KUKA KRL program: MyProgram_322().src

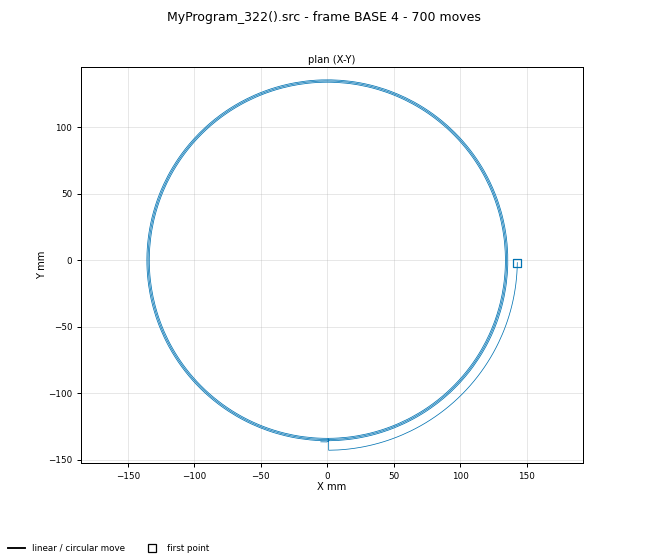
[picture p0: tool path of MyProgram_322().src in frame BASE 4, 700 of 700 moves have a stored position in this frame; points joined in program order, loops and branches not executed]
&ACCESS RVP
&REL 1
&PARAM TEMPLATE = C:\KRC\Roboter\Template\vorgabe
&PARAM EDITMASK = *
DEF MyProgram_322()
; ---- Setting reference (Base) ----
$BASE = BASE_DATA[4]

; --------------------------
; ---- Setting tool (TCP) ----
$TOOL = TOOL_DATA[3]
; --------------------------

$VEL.CP = VEL_APROX_PRINT
Startdeposition()
$VEL.CP = VEL_PRINT
LIN {X 142.7599,Y -1.7436,Z 185,A 2.3908,B 3.1922,C 0.193,E1 3.3578,E2 451.0051} C_DIS
LIN {X 142.6356,Y -6.2063,Z 185,A 0.7116,B 3.1919,C 0.1969,E1 3.3576,E2 452.6705} C_DIS
LIN {X 142.4407,Y -9.7017,Z 185,A -0.6684,B 3.1917,C 0.2006,E1 3.3574,E2 454.0481} C_DIS
LIN {X 142.1591,Y -13.1909,Z 185,A -2.1332,B 3.1914,C 0.2052,E1 3.357,E2 455.5219} C_DIS
LIN {X 141.6977,Y -17.466,Z 185,A -3.6398,B 3.1913,C 0.2077,E1 3.3566,E2 457.0004} C_DIS
LIN {X 141.2248,Y -20.9551,Z 185,A -4.9961,B 3.191,C 0.211,E1 3.356,E2 458.3501} C_DIS
LIN {X 140.669,Y -24.408,Z 185,A -6.3574,B 3.1908,C 0.2145,E1 3.3554,E2 459.7068} C_DIS
LIN {X 140.0285,Y -27.8456,Z 185,A -7.6988,B 3.1906,C 0.2178,E1 3.3547,E2 461.0409} C_DIS
LIN {X 139.3005,Y -31.2823,Z 185,A -9.0472,B 3.1904,C 0.221,E1 3.3539,E2 462.382} C_DIS
LIN {X 138.4934,Y -34.68,Z 185,A -10.3892,B 3.1901,C 0.2242,E1 3.353,E2 463.717} C_DIS
LIN {X 137.5957,Y -38.0853,Z 185,A -11.7403,B 3.1899,C 0.2274,E1 3.3521,E2 465.0608} C_DIS
LIN {X 136.4692,Y -41.9415,Z 185,A -13.3324,B 3.1896,C 0.2316,E1 3.3508,E2 466.6513} C_DIS
LIN {X 135.3217,Y -45.5096,Z 185,A -14.7313,B 3.1894,C 0.2346,E1 3.3496,E2 468.0371} C_DIS
LIN {X 134.1171,Y -48.9469,Z 185,A -16.135,B 3.1892,C 0.2379,E1 3.3483,E2 469.4342} C_DIS
LIN {X 132.912,Y -52.1294,Z 185,A -17.4464,B 3.1889,C 0.2409,E1 3.3469,E2 470.7393} C_DIS
LIN {X 131.5372,Y -55.5078,Z 185,A -18.8532,B 3.1887,C 0.2442,E1 3.3455,E2 472.1395} C_DIS
LIN {X 130.1671,Y -58.6477,Z 185,A -20.1759,B 3.1884,C 0.2472,E1 3.344,E2 473.4562} C_DIS
LIN {X 128.7579,Y -61.6788,Z 185,A -21.4838,B 3.1882,C 0.2503,E1 3.3424,E2 474.7605} C_DIS
LIN {X 126.9178,Y -65.3849,Z 185,A -23.0872,B 3.1879,C 0.254,E1 3.3404,E2 476.3576} C_DIS
LIN {X 124.8595,Y -69.2355,Z 185,A -24.7994,B 3.1876,C 0.258,E1 3.3381,E2 478.0657} C_DIS
LIN {X 122.6632,Y -73.0559,Z 185,A -26.5049,B 3.1873,C 0.2617,E1 3.3357,E2 479.7641} C_DIS
LIN {X 120.4066,Y -76.7189,Z 185,A -28.1924,B 3.187,C 0.2655,E1 3.3332,E2 481.4476} C_DIS
LIN {X 117.9943,Y -80.3801,Z 185,A -29.8939,B 3.1867,C 0.2692,E1 3.3306,E2 483.1427} C_DIS
LIN {X 115.4359,Y -84.0122,Z 185,A -31.5557,B 3.1864,C 0.2721,E1 3.3279,E2 484.7893} C_DIS
LIN {X 112.8442,Y -87.4622,Z 185,A -33.2618,B 3.1861,C 0.2758,E1 3.325,E2 486.4933} C_DIS
LIN {X 110.1935,Y -90.7797,Z 185,A -34.9543,B 3.1858,C 0.2796,E1 3.3221,E2 488.1855} C_DIS
LIN {X 107.2025,Y -94.293,Z 185,A -36.7037,B 3.1855,C 0.2826,E1 3.3189,E2 489.9224} C_DIS
LIN {X 104.325,Y -97.4668,Z 185,A -38.3639,B 3.1852,C 0.2857,E1 3.3158,E2 491.5759} C_DIS
LIN {X 101.2534,Y -100.6538,Z 185,A -40.0668,B 3.185,C 0.2887,E1 3.3124,E2 493.2702} C_DIS
LIN {X 98.1844,Y -103.65,Z 185,A -41.7616,B 3.1847,C 0.292,E1 3.309,E2 494.9627} C_DIS
LIN {X 94.9103,Y -106.6568,Z 185,A -43.4985,B 3.1844,C 0.295,E1 3.3054,E2 496.6945} C_DIS
LIN {X 91.5632,Y -109.5431,Z 185,A -45.1906,B 3.1841,C 0.2977,E1 3.3019,E2 498.3768} C_DIS
LIN {X 88.2302,Y -112.2447,Z 185,A -46.8727,B 3.1839,C 0.3005,E1 3.2982,E2 500.0548} C_DIS
LIN {X 84.7543,Y -114.8922,Z 185,A -48.591,B 3.1836,C 0.3033,E1 3.2944,E2 501.7696} C_DIS
LIN {X 81.1633,Y -117.457,Z 185,A -50.3222,B 3.1833,C 0.306,E1 3.2904,E2 503.4967} C_DIS
LIN {X 77.4935,Y -119.9095,Z 185,A -52.0213,B 3.1831,C 0.3082,E1 3.2865,E2 505.1871} C_DIS
LIN {X 73.8618,Y -122.1797,Z 185,A -53.6994,B 3.1829,C 0.3106,E1 3.2825,E2 506.8609} C_DIS
LIN {X 70.0297,Y -124.4158,Z 185,A -55.4462,B 3.1827,C 0.313,E1 3.2783,E2 508.6043} C_DIS
LIN {X 66.174,Y -126.5065,Z 185,A -57.1052,B 3.1825,C 0.3146,E1 3.2742,E2 510.2505} C_DIS
LIN {X 62.6225,Y -128.3029,Z 185,A -58.6591,B 3.1823,C 0.3164,E1 3.2703,E2 511.7996} C_DIS
LIN {X 59.4743,Y -129.7918,Z 185,A -59.9839,B 3.1823,C 0.3176,E1 3.267,E2 513.1153} C_DIS
LIN {X 56.3886,Y -131.1613,Z 185,A -61.3699,B 3.182,C 0.3196,E1 3.2634,E2 514.5065} C_DIS
LIN {X 52.762,Y -132.6631,Z 185,A -62.9943,B 3.1818,C 0.3219,E1 3.2592,E2 516.1389} C_DIS
LIN {X 48.9995,Y -134.0981,Z 185,A -64.5241,B 3.1817,C 0.323,E1 3.2552,E2 517.6578} C_DIS
LIN {X 45.7133,Y -135.2538,Z 185,A -65.8658,B 3.1816,C 0.324,E1 3.2517,E2 518.9926} C_DIS
LIN {X 42.3516,Y -136.3437,Z 185,A -67.3012,B 3.1814,C 0.3255,E1 3.2479,E2 520.4313} C_DIS
LIN {X 38.837,Y -137.3854,Z 185,A -68.8442,B 3.1812,C 0.3275,E1 3.2437,E2 521.9853} C_DIS
LIN {X 34.6802,Y -138.4934,Z 185,A -70.406,B 3.1812,C 0.3275,E1 3.2395,E2 523.5252} C_DIS
LIN {X 31.4204,Y -139.2689,Z 185,A -71.7456,B 3.1811,C 0.3286,E1 3.2359,E2 524.865} C_DIS
LIN {X 27.8611,Y -140.0253,Z 185,A -73.1737,B 3.1811,C 0.3294,E1 3.232,E2 526.2895} C_DIS
LIN {X 24.4235,Y -140.6662,Z 185,A -74.5592,B 3.1809,C 0.3302,E1 3.2282,E2 527.6734} C_DIS
LIN {X 20.03,Y -141.357,Z 185,A -76.38,B 3.1808,C 0.3315,E1 3.2231,E2 529.5001} C_DIS
LIN {X 15.7373,Y -141.8997,Z 185,A -78.0703,B 3.1808,C 0.332,E1 3.2184,E2 531.185} C_DIS
LIN {X 11.4541,Y -142.3099,Z 185,A -79.7619,B 3.1807,C 0.3324,E1 3.2137,E2 532.8726} C_DIS
LIN {X 7.9599,Y -142.5492,Z 185,A -81.1954,B 3.1807,C 0.3331,E1 3.2097,E2 534.3107} C_DIS
LIN {X 4.3071,Y -142.7045,Z 185,A -82.7592,B 3.1805,C 0.3343,E1 3.2053,E2 535.8887} C_DIS
LIN {X 1.005,Y -142.7647,Z 185,A -83.6736,B 3.1808,C 0.3313,E1 3.2029,E2 536.7463} C_DIS
Enddeposition()
LIN {X 0.9687,Y -133.816,Z 186,A -83.71,B 3.076,C 0.3108,E1 3.0971,E2 536.5076} C_DIS
Startdeposition()
$VEL.CP = VEL_PRINT
LIN {X 4.436,Y -133.7511,Z 186,A -81.8774,B 3.0763,C 0.3079,E1 3.1024,E2 534.6292} C_DIS
LIN {X 8.1929,Y -133.5716,Z 186,A -80.4113,B 3.0763,C 0.3084,E1 3.1064,E2 533.1809} C_DIS
LIN {X 11.4617,Y -133.331,Z 186,A -79.0228,B 3.0763,C 0.308,E1 3.1103,E2 531.7937} C_DIS
LIN {X 14.751,Y -133.0078,Z 186,A -77.6221,B 3.0763,C 0.3074,E1 3.1142,E2 530.394} C_DIS
LIN {X 18.5236,Y -132.5349,Z 186,A -75.9557,B 3.0765,C 0.3063,E1 3.1188,E2 528.7217} C_DIS
LIN {X 22.8645,Y -131.8567,Z 186,A -74.1261,B 3.0765,C 0.3055,E1 3.1238,E2 526.8978} C_DIS
LIN {X 26.0898,Y -131.2559,Z 186,A -72.7336,B 3.0766,C 0.3046,E1 3.1277,E2 525.506} C_DIS
LIN {X 29.3206,Y -130.5717,Z 186,A -71.3456,B 3.0767,C 0.3038,E1 3.1314,E2 524.1205} C_DIS
LIN {X 32.5132,Y -129.8133,Z 186,A -69.9613,B 3.0768,C 0.3028,E1 3.1352,E2 522.738} C_DIS
LIN {X 36.191,Y -128.8357,Z 186,A -68.2956,B 3.077,C 0.301,E1 3.1397,E2 521.0665} C_DIS
LIN {X 40.4049,Y -127.5772,Z 186,A -66.502,B 3.0771,C 0.2999,E1 3.1445,E2 519.2834} C_DIS
LIN {X 43.5438,Y -126.5402,Z 186,A -65.1143,B 3.0772,C 0.2986,E1 3.1481,E2 517.8983} C_DIS
LIN {X 47.1263,Y -125.2499,Z 186,A -63.5124,B 3.0774,C 0.297,E1 3.1523,E2 516.299} C_DIS
LIN {X 50.1812,Y -124.0574,Z 186,A -62.1351,B 3.0775,C 0.2956,E1 3.1559,E2 514.9243} C_DIS
LIN {X 53.7484,Y -122.556,Z 186,A -60.3934,B 3.0778,C 0.2928,E1 3.1604,E2 513.1704} C_DIS
LIN {X 57.6835,Y -120.7517,Z 186,A -58.6987,B 3.0778,C 0.2917,E1 3.1646,E2 511.495} C_DIS
LIN {X 60.1603,Y -119.5386,Z 186,A -57.5521,B 3.078,C 0.2903,E1 3.1675,E2 510.3521} C_DIS
LIN {X 63.3281,Y -117.8917,Z 186,A -56.1166,B 3.0781,C 0.2889,E1 3.171,E2 508.9276} C_DIS
LIN {X 66.3957,Y -116.1917,Z 186,A -54.5879,B 3.0784,C 0.2864,E1 3.1748,E2 507.3942} C_DIS
LIN {X 69.1892,Y -114.5502,Z 186,A -53.1474,B 3.0786,C 0.2838,E1 3.1782,E2 505.9457} C_DIS
LIN {X 72.8586,Y -112.252,Z 186,A -51.3975,B 3.0788,C 0.2817,E1 3.1823,E2 504.2079} C_DIS
LIN {X 76.0934,Y -110.0857,Z 186,A -49.6753,B 3.0791,C 0.2783,E1 3.1863,E2 502.4773} C_DIS
LIN {X 79.7248,Y -107.4845,Z 186,A -47.845,B 3.0794,C 0.2757,E1 3.1904,E2 500.6562} C_DIS
LIN {X 83.1812,Y -104.8324,Z 186,A -46.0377,B 3.0796,C 0.2728,E1 3.1944,E2 498.8549} C_DIS
LIN {X 86.574,Y -102.0483,Z 186,A -44.2223,B 3.0799,C 0.2698,E1 3.1983,E2 497.0463} C_DIS
LIN {X 89.8778,Y -99.1508,Z 186,A -42.4453,B 3.0801,C 0.267,E1 3.202,E2 495.2813} C_DIS
LIN {X 92.8686,Y -96.3556,Z 186,A -40.7416,B 3.0804,C 0.2639,E1 3.2054,E2 493.5826} C_DIS
LIN {X 95.7716,Y -93.4709,Z 186,A -38.9685,B 3.0807,C 0.2601,E1 3.2089,E2 491.8054} C_DIS
LIN {X 98.7809,Y -90.2849,Z 186,A -37.1738,B 3.081,C 0.2568,E1 3.2123,E2 490.0196} C_DIS
LIN {X 101.6976,Y -86.9865,Z 186,A -35.4113,B 3.0812,C 0.2538,E1 3.2155,E2 488.2715} C_DIS
LIN {X 104.127,Y -84.0623,Z 186,A -33.8119,B 3.0815,C 0.2504,E1 3.2183,E2 486.6744} C_DIS
LIN {X 106.8292,Y -80.6004,Z 186,A -31.9916,B 3.0818,C 0.2466,E1 3.2214,E2 484.8602} C_DIS
LIN {X 109.4259,Y -77.0383,Z 186,A -30.1807,B 3.0821,C 0.2429,E1 3.2243,E2 483.0577} C_DIS
LIN {X 111.8951,Y -73.406,Z 186,A -28.3662,B 3.0824,C 0.239,E1 3.2272,E2 481.2502} C_DIS
LIN {X 113.9323,Y -70.2026,Z 186,A -26.9035,B 3.0826,C 0.2366,E1 3.2293,E2 479.8069} C_DIS
LIN {X 115.8253,Y -67.0328,Z 186,A -25.3615,B 3.0829,C 0.2331,E1 3.2315,E2 478.2686} C_DIS
LIN {X 117.4797,Y -64.0892,Z 186,A -23.9557,B 3.0831,C 0.2299,E1 3.2334,E2 476.8668} C_DIS
LIN {X 119.0131,Y -61.1926,Z 186,A -22.6488,B 3.0833,C 0.2272,E1 3.235,E2 475.571} C_DIS
LIN {X 120.2635,Y -58.6973,Z 186,A -21.492,B 3.0835,C 0.2245,E1 3.2365,E2 474.4182} C_DIS
LIN {X 121.6664,Y -55.7303,Z 186,A -20.0767,B 3.0838,C 0.2208,E1 3.2381,E2 473.0004} C_DIS
LIN {X 123.431,Y -51.7028,Z 186,A -18.256,B 3.0841,C 0.2165,E1 3.2401,E2 471.1861} C_DIS
LIN {X 124.9906,Y -47.8147,Z 186,A -16.4578,B 3.0844,C 0.2117,E1 3.242,E2 469.386} C_DIS
LIN {X 126.1657,Y -44.6236,Z 186,A -15.0773,B 3.0846,C 0.2085,E1 3.2432,E2 468.014} C_DIS
LIN {X 127.5813,Y -40.3922,Z 186,A -13.3493,B 3.0849,C 0.2051,E1 3.2447,E2 466.3077} C_DIS
LIN {X 128.8337,Y -36.1982,Z 186,A -11.5227,B 3.0852,C 0.2005,E1 3.2461,E2 464.4856} C_DIS
LIN {X 129.9409,Y -32.0037,Z 186,A -9.8212,B 3.0854,C 0.1969,E1 3.2473,E2 462.8025} C_DIS
LIN {X 130.6882,Y -28.7984,Z 186,A -8.4768,B 3.0856,C 0.1937,E1 3.2481,E2 461.4653} C_DIS
LIN {X 131.3542,Y -25.5879,Z 186,A -7.1334,B 3.0858,C 0.1904,E1 3.2489,E2 460.1284} C_DIS
LIN {X 131.9414,Y -22.3615,Z 186,A -5.9696,B 3.0859,C 0.1888,E1 3.2494,E2 458.9938} C_DIS
LIN {X 132.3756,Y -19.6384,Z 186,A -4.5318,B 3.0863,C 0.183,E1 3.25,E2 457.5229} C_DIS
LIN {X 132.8782,Y -15.8696,Z 186,A -3.1128,B 3.0863,C 0.1805,E1 3.2505,E2 456.1289} C_DIS
LIN {X 133.2421,Y -12.4557,Z 186,A -1.7289,B 3.0866,C 0.1772,E1 3.2509,E2 454.7548} C_DIS
LIN {X 133.4983,Y -9.3201,Z 186,A -0.4325,B 3.0868,C 0.1739,E1 3.2512,E2 453.4639} C_DIS
LIN {X 133.7115,Y -5.4589,Z 186,A 1.2482,B 3.087,C 0.169,E1 3.2514,E2 451.7789} C_DIS
LIN {X 133.8137,Y -1.6575,Z 186,A 2.6544,B 3.0872,C 0.1666,E1 3.2514,E2 450.3995} C_DIS
LIN {X 133.805,Y 2.1748,Z 186,A 4.3608,B 3.0875,C 0.1613,E1 3.2514,E2 448.6837} C_DIS
LIN {X 133.6617,Y 6.5635,Z 186,A 6.0882,B 3.0877,C 0.1575,E1 3.2512,E2 446.9743} C_DIS
LIN {X 133.4607,Y 9.8358,Z 186,A 7.4615,B 3.0878,C 0.1539,E1 3.251,E2 445.6039} C_DIS
LIN {X 133.1787,Y 13.1156,Z 186,A 8.766,B 3.088,C 0.1509,E1 3.2506,E2 444.3115} C_DIS
LIN {X 132.8167,Y 16.3854,Z 186,A 10.2269,B 3.0882,C 0.1465,E1 3.2502,E2 442.8433} C_DIS
LIN {X 132.2965,Y 20.154,Z 186,A 11.5023,B 3.0882,C 0.1454,E1 3.2497,E2 441.6108} C_DIS
LIN {X 131.855,Y 22.8737,Z 186,A 12.8158,B 3.0885,C 0.1408,E1 3.2491,E2 440.2802} C_DIS
LIN {X 131.2542,Y 26.0985,Z 186,A 14.1611,B 3.0886,C 0.1375,E1 3.2484,E2 438.9414} C_DIS
LIN {X 130.571,Y 29.3235,Z 186,A 15.5046,B 3.0888,C 0.1343,E1 3.2476,E2 437.6055} C_DIS
LIN {X 129.8121,Y 32.5177,Z 186,A 16.8476,B 3.0888,C 0.131,E1 3.2467,E2 436.2695} C_DIS
LIN {X 128.8341,Y 36.1967,Z 186,A 18.466,B 3.0891,C 0.1267,E1 3.2455,E2 434.6516} C_DIS
LIN {X 127.5731,Y 40.418,Z 186,A 20.3118,B 3.0893,C 0.122,E1 3.244,E2 432.81} C_DIS
LIN {X 126.1683,Y 44.6162,Z 186,A 22.1632,B 3.0894,C 0.1173,E1 3.2423,E2 430.9631} C_DIS
LIN {X 124.6797,Y 48.6144,Z 186,A 23.7847,B 3.0895,C 0.1145,E1 3.2407,E2 429.366} C_DIS
LIN {X 123.4332,Y 51.6976,Z 186,A 25.2113,B 3.0897,C 0.1107,E1 3.2392,E2 427.9385} C_DIS
LIN {X 121.6698,Y 55.723,Z 186,A 27.062,B 3.0898,C 0.1061,E1 3.2371,E2 426.0909} C_DIS
LIN {X 120.0375,Y 59.1553,Z 186,A 28.3574,B 3.0898,C 0.1051,E1 3.2355,E2 424.8353} C_DIS
LIN {X 118.7857,Y 61.634,Z 186,A 29.6269,B 3.09,C 0.1013,E1 3.2339,E2 423.5556} C_DIS
LIN {X 117.2392,Y 64.529,Z 186,A 31.1268,B 3.0901,C 0.0969,E1 3.2319,E2 422.0437} C_DIS
LIN {X 115.3504,Y 67.8467,Z 186,A 32.5705,B 3.0902,C 0.0947,E1 3.2299,E2 420.6227} C_DIS
LIN {X 113.3422,Y 71.1516,Z 186,A 34.2658,B 3.0903,C 0.0903,E1 3.2274,E2 418.922} C_DIS
LIN {X 111.2743,Y 74.3434,Z 186,A 35.729,B 3.0904,C 0.0879,E1 3.2252,E2 417.4784} C_DIS
LIN {X 109.4199,Y 77.0468,Z 186,A 37.1703,B 3.0905,C 0.0843,E1 3.2229,E2 416.0322} C_DIS
LIN {X 106.8195,Y 80.6133,Z 186,A 39.0047,B 3.0906,C 0.0805,E1 3.2198,E2 414.2041} C_DIS
LIN {X 103.9631,Y 84.2655,Z 186,A 40.926,B 3.0907,C 0.0766,E1 3.2165,E2 412.29} C_DIS
LIN {X 101.1608,Y 87.61,Z 186,A 42.7319,B 3.0908,C 0.073,E1 3.2132,E2 410.4913} C_DIS
LIN {X 98.4298,Y 90.6669,Z 186,A 44.4122,B 3.0908,C 0.07,E1 3.2101,E2 408.8197} C_DIS
LIN {X 95.582,Y 93.6641,Z 186,A 46.1113,B 3.0909,C 0.0669,E1 3.2068,E2 407.1289} C_DIS
LIN {X 92.473,Y 96.7349,Z 186,A 47.8811,B 3.091,C 0.064,E1 3.2033,E2 405.371} C_DIS
LIN {X 89.6931,Y 99.3184,Z 186,A 49.5251,B 3.091,C 0.0606,E1 3.1999,E2 403.7246} C_DIS
LIN {X 86.5877,Y 102.0367,Z 186,A 51.2202,B 3.0911,C 0.0579,E1 3.1963,E2 402.0379} C_DIS
LIN {X 83.1898,Y 104.8255,Z 186,A 53.0445,B 3.0911,C 0.0549,E1 3.1924,E2 400.2205} C_DIS
LIN {X 79.7194,Y 107.4885,Z 186,A 54.8692,B 3.0912,C 0.052,E1 3.1883,E2 398.4015} C_DIS
LIN {X 76.2646,Y 109.9666,Z 186,A 56.4511,B 3.0912,C 0.0509,E1 3.1848,E2 396.8481} C_DIS
LIN {X 73.4139,Y 111.8899,Z 186,A 58.0702,B 3.0913,C 0.0473,E1 3.181,E2 395.2115} C_DIS
LIN {X 70.2047,Y 113.931,Z 186,A 59.555,B 3.0913,C 0.0459,E1 3.1775,E2 393.7439} C_DIS
LIN {X 67.3921,Y 115.6173,Z 186,A 61.0498,B 3.0913,C 0.043,E1 3.1739,E2 392.2383} C_DIS
LIN {X 64.0999,Y 117.4739,Z 186,A 62.5393,B 3.0913,C 0.0417,E1 3.1703,E2 390.7642} C_DIS
LIN {X 61.1645,Y 119.0273,Z 186,A 63.7829,B 3.0913,C 0.0411,E1 3.1672,E2 389.542} C_DIS
LIN {X 58.6915,Y 120.2663,Z 186,A 65.0633,B 3.0914,C 0.0388,E1 3.164,E2 388.2503} C_DIS
LIN {X 55.7246,Y 121.6691,Z 186,A 66.5094,B 3.0914,C 0.0367,E1 3.1603,E2 386.7994} C_DIS
LIN {X 51.6992,Y 123.4325,Z 186,A 68.3671,B 3.0914,C 0.0346,E1 3.1555,E2 384.9448} C_DIS
LIN {X 48.1677,Y 124.8534,Z 186,A 69.8792,B 3.0914,C 0.0336,E1 3.1516,E2 383.447} C_DIS
LIN {X 44.6082,Y 126.1712,Z 186,A 71.6386,B 3.0915,C 0.0309,E1 3.147,E2 381.6721} C_DIS
LIN {X 40.9108,Y 127.4156,Z 186,A 72.9052,B 3.0915,C 0.0323,E1 3.1437,E2 380.4535} C_DIS
LIN {X 38.341,Y 128.2145,Z 186,A 74.4123,B 3.0915,C 0.0286,E1 3.1396,E2 378.9047} C_DIS
LIN {X 34.1077,Y 129.4034,Z 186,A 76.1827,B 3.0915,C 0.0278,E1 3.1349,E2 377.1481} C_DIS
LIN {X 30.4151,Y 130.3217,Z 186,A 77.7251,B 3.0915,C 0.0271,E1 3.1307,E2 375.6164} C_DIS
LIN {X 27.2108,Y 131.0279,Z 186,A 79.1175,B 3.0915,C 0.0262,E1 3.1269,E2 374.2259} C_DIS
LIN {X 23.9747,Y 131.658,Z 186,A 80.5085,B 3.0915,C 0.0255,E1 3.1231,E2 372.8377} C_DIS
LIN {X 21.261,Y 132.125,Z 186,A 81.6808,B 3.0915,C 0.0249,E1 3.1199,E2 371.6666} C_DIS
LIN {X 17.4962,Y 132.6739,Z 186,A 83.2879,B 3.0915,C 0.0242,E1 3.1154,E2 370.0626} C_DIS
LIN {X 14.2377,Y 133.063,Z 186,A 84.6779,B 3.0915,C 0.0237,E1 3.1116,E2 368.6748} C_DIS
LIN {X 10.7215,Y 133.3935,Z 186,A 86.1554,B 3.0915,C 0.0234,E1 3.1075,E2 367.202} C_DIS
LIN {X 7.6847,Y 133.6029,Z 186,A 87.6138,B 3.0915,C 0.0219,E1 3.1033,E2 365.7258} C_DIS
LIN {X 3.2935,Y 133.7828,Z 186,A 89.4572,B 3.0915,C 0.0218,E1 3.0982,E2 363.8877} C_DIS
LIN {X 0.0194,Y 133.8247,Z 186,A 90.9014,B 3.0915,C 0.0213,E1 3.0941,E2 362.4391} C_DIS
LIN {X -3.8109,Y 133.7684,Z 186,A 92.3893,B 3.0915,C 0.0222,E1 3.09,E2 360.9698} C_DIS
LIN {X -7.6749,Y 133.6035,Z 186,A 94.1786,B 3.0915,C 0.0214,E1 3.085,E2 359.1656} C_DIS
LIN {X -11.4718,Y 133.3301,Z 186,A 95.6768,B 3.0915,C 0.0224,E1 3.0809,E2 357.6837} C_DIS
LIN {X -14.735,Y 133.0095,Z 186,A 97.2161,B 3.0915,C 0.0218,E1 3.0765,E2 356.129} C_DIS
LIN {X -18.5315,Y 132.5338,Z 186,A 98.7427,B 3.0915,C 0.0229,E1 3.0724,E2 354.6164} C_DIS
LIN {X -21.2546,Y 132.1261,Z 186,A 99.9336,B 3.0915,C 0.0232,E1 3.0691,E2 353.4248} C_DIS
LIN {X -24.4869,Y 131.5647,Z 186,A 101.3433,B 3.0915,C 0.0237,E1 3.0652,E2 352.0152} C_DIS
LIN {X -27.7046,Y 130.9244,Z 186,A 102.7609,B 3.0915,C 0.0243,E1 3.0613,E2 350.5968} C_DIS
LIN {X -30.9214,Y 130.2017,Z 186,A 104.1784,B 3.0915,C 0.025,E1 3.0574,E2 349.1794} C_DIS
LIN {X -34.1058,Y 129.4038,Z 186,A 105.7068,B 3.0915,C 0.025,E1 3.0533,E2 347.6372} C_DIS
LIN {X -38.3371,Y 128.2157,Z 186,A 107.6473,B 3.0915,C 0.026,E1 3.048,E2 345.6909} C_DIS
LIN {X -42.4834,Y 126.8999,Z 186,A 109.4445,B 3.0915,C 0.0278,E1 3.0433,E2 343.9025} C_DIS
LIN {X -46.6119,Y 125.4426,Z 186,A 111.3916,B 3.0915,C 0.029,E1 3.0381,E2 341.948} C_DIS
LIN {X -50.1272,Y 124.0792,Z 186,A 112.921,B 3.0915,C 0.031,E1 3.0342,E2 340.4297} C_DIS
LIN {X -53.6243,Y 122.6096,Z 186,A 114.7123,B 3.0915,C 0.0317,E1 3.0295,E2 338.6197} C_DIS
LIN {X -57.6877,Y 120.7497,Z 186,A 116.5245,B 3.0915,C 0.0343,E1 3.025,E2 336.8207} C_DIS
LIN {X -60.1639,Y 119.5368,Z 186,A 117.7263,B 3.0915,C 0.0356,E1 3.022,E2 335.6171} C_DIS
LIN {X -63.091,Y 118.0191,Z 186,A 119.1641,B 3.0915,C 0.0372,E1 3.0184,E2 334.1772} C_DIS
LIN {X -66.4175,Y 116.1793,Z 186,A 120.8328,B 3.0915,C 0.0391,E1 3.0143,E2 332.5047} C_DIS
LIN {X -69.2409,Y 114.519,Z 186,A 122.3711,B 3.0915,C 0.0403,E1 3.0106,E2 330.9513} C_DIS
LIN {X -72.9631,Y 112.1842,Z 186,A 124.1948,B 3.0914,C 0.0433,E1 3.0063,E2 329.1357} C_DIS
LIN {X -75.6888,Y 110.3635,Z 186,A 125.6379,B 3.0914,C 0.0452,E1 3.003,E2 327.6889} C_DIS
LIN {X -78.8051,Y 108.1608,Z 186,A 127.432,B 3.0914,C 0.047,E1 2.9989,E2 325.8769} C_DIS
LIN {X -82.2857,Y 105.5373,Z 186,A 129.3446,B 3.0913,C 0.0499,E1 2.9946,E2 323.9602} C_DIS
LIN {X -85.4219,Y 103.0145,Z 186,A 131.0248,B 3.0913,C 0.053,E1 2.991,E2 322.2864} C_DIS
LIN {X -88.429,Y 100.4455,Z 186,A 132.8137,B 3.0912,C 0.0556,E1 2.9872,E2 320.4873} C_DIS
LIN {X -91.2759,Y 97.8652,Z 186,A 134.5475,B 3.0912,C 0.0582,E1 2.9836,E2 318.7442} C_DIS
LIN {X -94.5247,Y 94.7315,Z 186,A 136.4745,B 3.091,C 0.062,E1 2.9798,E2 316.8193} C_DIS
LIN {X -97.4999,Y 91.6663,Z 186,A 138.3685,B 3.091,C 0.0653,E1 2.9761,E2 314.9189} C_DIS
LIN {X -100.2187,Y 88.6855,Z 186,A 140.2061,B 3.091,C 0.0684,E1 2.9727,E2 313.0695} C_DIS
LIN {X -102.7756,Y 85.7102,Z 186,A 141.9342,B 3.0908,C 0.0717,E1 2.9695,E2 311.3369} C_DIS
LIN {X -105.3432,Y 82.5333,Z 186,A 143.7165,B 3.0908,C 0.0754,E1 2.9664,E2 309.5519} C_DIS
LIN {X -107.4874,Y 79.7209,Z 186,A 145.3525,B 3.0907,C 0.0782,E1 2.9637,E2 307.9024} C_DIS
LIN {X -109.7041,Y 76.6418,Z 186,A 146.9268,B 3.0906,C 0.0821,E1 2.9611,E2 306.3354} C_DIS
LIN {X -111.8681,Y 73.447,Z 186,A 148.7552,B 3.0905,C 0.0852,E1 2.9583,E2 304.4871} C_DIS
LIN {X -113.9334,Y 70.2007,Z 186,A 150.3614,B 3.0904,C 0.0893,E1 2.9559,E2 302.887} C_DIS
LIN {X -115.6194,Y 67.3885,Z 186,A 151.9478,B 3.0903,C 0.0919,E1 2.9536,E2 301.2798} C_DIS
LIN {X -117.4869,Y 64.0759,Z 186,A 153.6452,B 3.0902,C 0.0957,E1 2.9513,E2 299.5752} C_DIS
LIN {X -119.0224,Y 61.1743,Z 186,A 155.0004,B 3.0901,C 0.0993,E1 2.9496,E2 298.2272} C_DIS
LIN {X -120.2643,Y 58.6956,Z 186,A 156.2361,B 3.09,C 0.1021,E1 2.948,E2 296.9865} C_DIS
LIN {X -121.6724,Y 55.7174,Z 186,A 157.7877,B 3.0899,C 0.1052,E1 2.9462,E2 295.4189} C_DIS
LIN {X -123.4363,Y 51.6902,Z 186,A 159.7632,B 3.0897,C 0.1097,E1 2.944,E2 293.4334} C_DIS
LIN {X -124.8557,Y 48.1618,Z 186,A 161.373,B 3.0896,C 0.114,E1 2.9424,E2 291.8272} C_DIS
LIN {X -126.1752,Y 44.5967,Z 186,A 163.25,B 3.0894,C 0.1174,E1 2.9406,E2 289.9211} C_DIS
LIN {X -127.5735,Y 40.4167,Z 186,A 165.1043,B 3.0892,C 0.1226,E1 2.939,E2 288.0722} C_DIS
LIN {X -128.829,Y 36.2149,Z 186,A 167.1441,B 3.0891,C 0.1271,E1 2.9374,E2 286.014} C_DIS
LIN {X -129.9288,Y 32.0536,Z 186,A 168.9334,B 3.0888,C 0.1323,E1 2.9361,E2 284.2327} C_DIS
LIN {X -130.6486,Y 28.9817,Z 186,A 170.4857,B 3.0888,C 0.1353,E1 2.9352,E2 282.6566} C_DIS
LIN {X -131.3576,Y 25.5702,Z 186,A 171.9247,B 3.0885,C 0.1396,E1 2.9344,E2 281.2252} C_DIS
LIN {X -131.9416,Y 22.36,Z 186,A 173.2095,B 3.0883,C 0.1439,E1 2.9338,E2 279.955} C_DIS
LIN {X -132.3758,Y 19.6369,Z 186,A 174.7809,B 3.0883,C 0.1458,E1 2.9331,E2 278.3367} C_DIS
LIN {X -132.8802,Y 15.853,Z 186,A 176.3395,B 3.088,C 0.1506,E1 2.9325,E2 276.7885} C_DIS
LIN {X -133.2292,Y 12.5891,Z 186,A 177.8078,B 3.0878,C 0.1543,E1 2.9321,E2 275.3134} C_DIS
LIN {X -133.4984,Y 9.3193,Z 186,A 179.2738,B 3.0876,C 0.1581,E1 2.9318,E2 273.8408} C_DIS
LIN {X -133.7116,Y 5.4557,Z 186,A -178.8777,B 3.0874,C 0.1621,E1 2.9316,E2 271.9698} C_DIS
LIN {X -133.8185,Y 1.1931,Z 186,A -177.0341,B 3.0871,C 0.1671,E1 2.9315,E2 270.1252} C_DIS
LIN {X -133.7956,Y -2.7401,Z 186,A -175.1638,B 3.0869,C 0.1712,E1 2.9315,E2 268.2329} C_DIS
LIN {X -133.6337,Y -7.1206,Z 186,A -173.2113,B 3.0866,C 0.1762,E1 2.9318,E2 266.2721} C_DIS
LIN {X -133.3293,Y -11.4813,Z 186,A -171.3647,B 3.0863,C 0.1816,E1 2.9322,E2 264.4298} C_DIS
LIN {X -133.0076,Y -14.7528,Z 186,A -169.8935,B 3.0861,C 0.1853,E1 2.9326,E2 262.9516} C_DIS
LIN {X -132.534,Y -18.5298,Z 186,A -168.1657,B 3.0859,C 0.1895,E1 2.9333,E2 261.2125} C_DIS
LIN {X -132.1258,Y -21.256,Z 186,A -166.9237,B 3.0857,C 0.1925,E1 2.9338,E2 259.9635} C_DIS
LIN {X -131.5619,Y -24.5012,Z 186,A -165.4497,B 3.0854,C 0.1962,E1 2.9345,E2 258.4823} C_DIS
LIN {X -130.921,Y -27.72,Z 186,A -163.9799,B 3.0852,C 0.1998,E1 2.9354,E2 257.0052} C_DIS
LIN {X -130.2015,Y -30.9224,Z 186,A -162.51,B 3.085,C 0.2034,E1 2.9363,E2 255.5279} C_DIS
LIN {X -129.4038,Y -34.1058,Z 186,A -160.9176,B 3.0848,C 0.2065,E1 2.9374,E2 253.9128} C_DIS
LIN {X -128.2198,Y -38.323,Z 186,A -158.9387,B 3.0845,C 0.2112,E1 2.939,E2 251.9219} C_DIS
LIN {X -126.9457,Y -42.3459,Z 186,A -157.0966,B 3.0841,C 0.2158,E1 2.9406,E2 250.0761} C_DIS
LIN {X -125.4386,Y -46.6225,Z 186,A -155.0454,B 3.0838,C 0.2205,E1 2.9425,E2 248.0121} C_DIS
LIN {X -124.0587,Y -50.1782,Z 186,A -153.452,B 3.0835,C 0.2249,E1 2.9442,E2 246.4244} C_DIS
LIN {X -122.5566,Y -53.7468,Z 186,A -151.5943,B 3.0832,C 0.2283,E1 2.9463,E2 244.5421} C_DIS
LIN {X -120.7471,Y -57.6932,Z 186,A -149.7824,B 3.0829,C 0.2332,E1 2.9484,E2 242.7369} C_DIS
LIN {X -119.5333,Y -60.1707,Z 186,A -148.5552,B 3.0827,C 0.2359,E1 2.9499,E2 241.5044} C_DIS
LIN {X -118.0212,Y -63.0871,Z 186,A -147.0903,B 3.0824,C 0.2391,E1 2.9518,E2 240.0326} C_DIS
LIN {X -116.1872,Y -66.4037,Z 186,A -145.3525,B 3.0821,C 0.2426,E1 2.9542,E2 238.2808} C_DIS
LIN {X -114.5139,Y -69.2492,Z 186,A -143.8159,B 3.0819,C 0.2454,E1 2.9565,E2 236.729} C_DIS
LIN {X -112.1775,Y -72.9734,Z 186,A -141.9641,B 3.0816,C 0.2499,E1 2.9592,E2 234.8817} C_DIS
LIN {X -110.354,Y -75.7026,Z 186,A -140.5047,B 3.0813,C 0.2528,E1 2.9615,E2 233.4158} C_DIS
LIN {X -108.1418,Y -78.8313,Z 186,A -138.6741,B 3.0811,C 0.2556,E1 2.9646,E2 231.5614} C_DIS
LIN {X -105.4975,Y -82.3367,Z 186,A -136.7271,B 3.0808,C 0.2594,E1 2.9679,E2 229.6063} C_DIS
LIN {X -102.9241,Y -85.5312,Z 186,A -134.9926,B 3.0805,C 0.2632,E1 2.971,E2 227.8749} C_DIS
LIN {X -100.6243,Y -88.2256,Z 186,A -133.3439,B 3.0802,C 0.2657,E1 2.974,E2 226.2096} C_DIS
LIN {X -97.8648,Y -91.2764,Z 186,A -131.539,B 3.08,C 0.269,E1 2.9774,E2 224.3994} C_DIS
LIN {X -95.0244,Y -94.2299,Z 186,A -129.7285,B 3.0797,C 0.2721,E1 2.981,E2 222.582} C_DIS
LIN {X -91.821,Y -97.354,Z 186,A -127.7762,B 3.0794,C 0.2754,E1 2.9849,E2 220.6252} C_DIS
LIN {X -88.6479,Y -100.2519,Z 186,A -125.8625,B 3.0791,C 0.2784,E1 2.9889,E2 218.7022} C_DIS
LIN {X -85.5342,Y -102.9216,Z 186,A -124.0928,B 3.0789,C 0.2813,E1 2.9927,E2 216.9308} C_DIS
LIN {X -82.3401,Y -105.4949,Z 186,A -122.2216,B 3.0786,C 0.2836,E1 2.9968,E2 215.045} C_DIS
LIN {X -78.8112,Y -108.1564,Z 186,A -120.2903,B 3.0784,C 0.2863,E1 3.0012,E2 213.1086} C_DIS
LIN {X -75.273,Y -110.648,Z 186,A -118.3822,B 3.0782,C 0.2888,E1 3.0056,E2 211.1934} C_DIS
LIN {X -71.5985,Y -113.0601,Z 186,A -116.5793,B 3.0779,C 0.2918,E1 3.0098,E2 209.4007} C_DIS
LIN {X -68.8002,Y -114.7848,Z 186,A -115.1158,B 3.0777,C 0.2934,E1 3.0133,E2 207.9298} C_DIS
LIN {X -65.5286,Y -116.6829,Z 186,A -113.477,B 3.0775,C 0.2953,E1 3.0173,E2 206.2883} C_DIS
LIN {X -62.6225,Y -118.2666,Z 186,A -111.9578,B 3.0775,C 0.2964,E1 3.0211,E2 204.7558} C_DIS
LIN {X -59.1648,Y -120.0328,Z 186,A -110.2662,B 3.0773,C 0.2981,E1 3.0253,E2 203.0601} C_DIS
LIN {X -55.7275,Y -121.6677,Z 186,A -108.6079,B 3.0771,C 0.2997,E1 3.0295,E2 201.3979} C_DIS
LIN {X -51.7027,Y -123.431,Z 186,A -106.6811,B 3.077,C 0.3012,E1 3.0345,E2 199.4649} C_DIS
LIN {X -48.1691,Y -124.8528,Z 186,A -105.0798,B 3.0768,C 0.3028,E1 3.0386,E2 197.867} C_DIS
LIN {X -44.582,Y -126.1803,Z 186,A -103.2946,B 3.0768,C 0.3032,E1 3.0434,E2 196.0624} C_DIS
LIN {X -40.4139,Y -127.5743,Z 186,A -101.4971,B 3.0766,C 0.3051,E1 3.0481,E2 194.2753} C_DIS
LIN {X -36.1998,Y -128.8333,Z 186,A -99.5276,B 3.0766,C 0.3057,E1 3.0535,E2 192.2941} C_DIS
LIN {X -32.0111,Y -129.9391,Z 186,A -97.7747,B 3.0764,C 0.3074,E1 3.0582,E2 190.554} C_DIS
LIN {X -28.4924,Y -130.7543,Z 186,A -96.3132,B 3.0762,C 0.3086,E1 3.0621,E2 189.103} C_DIS
LIN {X -25.5925,Y -131.3533,Z 186,A -94.9394,B 3.0762,C 0.3084,E1 3.0659,E2 187.7149} C_DIS
LIN {X -21.2653,Y -132.1243,Z 186,A -93.0461,B 3.0762,C 0.3089,E1 3.0712,E2 185.8196} C_DIS
LIN {X -17.4997,Y -132.6734,Z 186,A -91.4179,B 3.0762,C 0.3093,E1 3.0757,E2 184.1908} C_DIS
LIN {X -14.222,Y -133.0647,Z 186,A -90.006,B 3.0762,C 0.3095,E1 3.0796,E2 182.7785} C_DIS
LIN {X -10.9608,Y -133.3733,Z 186,A -88.6077,B 3.0762,C 0.3097,E1 3.0835,E2 181.3802} C_DIS
LIN {X -7.6949,Y -133.6023,Z 186,A -87.0658,B 3.0762,C 0.3087,E1 3.0879,E2 179.8195} C_DIS
LIN {X -3.3037,Y -133.7825,Z 186,A -85.2191,B 3.0762,C 0.3087,E1 3.093,E2 177.9765} C_DIS
LIN {X 0.005,Y -133.8247,Z 186,A -83.7567,B 3.0762,C 0.3082,E1 3.0971,E2 176.5075} C_DIS
LIN {X 0.005,Y -133.8247,Z 186,A -83.7567,B 3.0762,C 0.3082,E1 3.0971,E2 176.5075} C_DIS
Enddeposition()
LIN {X 0.9798,Y -134.7172,Z 186,A -83.5222,B 3.076,C 0.3111,E1 3.0977,E2 176.3268} C_DIS
Startdeposition()
$VEL.CP = VEL_PRINT
LIN {X -4.7209,Y -134.6408,Z 186,A -86.3903,B 3.0757,C 0.3146,E1 3.0895,E2 179.2542} C_DIS
LIN {X -9.5556,Y -134.3834,Z 186,A -88.596,B 3.0756,C 0.3156,E1 3.0833,E2 181.4799} C_DIS
LIN {X -13.4972,Y -134.0461,Z 186,A -90.522,B 3.0754,C 0.3171,E1 3.0778,E2 183.4382} C_DIS
LIN {X -17.9446,Y -133.5227,Z 186,A -92.1116,B 3.0757,C 0.3147,E1 3.0735,E2 184.9876} C_DIS
LIN {X -20.9348,Y -133.0862,Z 186,A -93.4283,B 3.0757,C 0.3145,E1 3.0699,E2 186.3089} C_DIS
LIN {X -24.4626,Y -132.4848,Z 186,A -94.9615,B 3.0757,C 0.3141,E1 3.0656,E2 187.8442} C_DIS
LIN {X -27.0994,Y -131.9688,Z 186,A -96.125,B 3.0757,C 0.3138,E1 3.0624,E2 189.0107} C_DIS
LIN {X -30.6293,Y -131.1958,Z 186,A -97.7819,B 3.0757,C 0.3138,E1 3.0579,E2 190.6837} C_DIS
LIN {X -34.4517,Y -130.2429,Z 186,A -99.439,B 3.0759,C 0.3129,E1 3.0534,E2 192.3389} C_DIS
LIN {X -38.5932,Y -129.0783,Z 186,A -101.2099,B 3.076,C 0.3114,E1 3.0487,E2 194.1027} C_DIS
LIN {X -41.1843,Y -128.2729,Z 186,A -102.4115,B 3.076,C 0.3109,E1 3.0454,E2 195.3108} C_DIS
LIN {X -44.2442,Y -127.2498,Z 186,A -103.7685,B 3.0762,C 0.3097,E1 3.0418,E2 196.6661} C_DIS
LIN {X -47.6042,Y -126.0318,Z 186,A -105.3267,B 3.0762,C 0.3087,E1 3.0377,E2 198.2296} C_DIS
LIN {X -51.3118,Y -124.5695,Z 186,A -107.1343,B 3.0764,C 0.3079,E1 3.033,E2 200.0521} C_DIS
LIN {X -55.0097,Y -122.9794,Z 186,A -108.836,B 3.0765,C 0.3061,E1 3.0287,E2 201.7527} C_DIS
LIN {X -58.6982,Y -121.2642,Z 186,A -110.5258,B 3.0767,C 0.3041,E1 3.0244,E2 203.4376} C_DIS
LIN {X -61.5273,Y -119.8524,Z 186,A -111.947,B 3.0768,C 0.303,E1 3.0208,E2 204.8688} C_DIS
LIN {X -65.4124,Y -117.7786,Z 186,A -114.2009,B 3.0768,C 0.3028,E1 3.0152,E2 207.1719} C_DIS
LIN {X -68.6164,Y -115.9419,Z 186,A -115.5415,B 3.0772,C 0.2995,E1 3.012,E2 208.4832} C_DIS
LIN {X -72.1199,Y -113.7951,Z 186,A -117.326,B 3.0774,C 0.2973,E1 3.0078,E2 210.2725} C_DIS
LIN {X -75.9221,Y -111.2948,Z 186,A -119.282,B 3.0777,C 0.2947,E1 3.0032,E2 212.2312} C_DIS
LIN {X -79.2603,Y -108.9423,Z 186,A -121.0384,B 3.0779,C 0.2921,E1 2.9992,E2 213.9901} C_DIS
LIN {X -82.7787,Y -106.2936,Z 186,A -122.9946,B 3.0781,C 0.2896,E1 2.9949,E2 215.9569} C_DIS
LIN {X -86.264,Y -103.4856,Z 186,A -124.9923,B 3.0784,C 0.2869,E1 2.9905,E2 217.9666} C_DIS
LIN {X -89.6696,Y -100.5484,Z 186,A -126.9122,B 3.0787,C 0.2835,E1 2.9865,E2 219.8873} C_DIS
LIN {X -92.8097,Y -97.6578,Z 186,A -128.8442,B 3.0789,C 0.2808,E1 2.9825,E2 221.8339} C_DIS
LIN {X -95.977,Y -94.5466,Z 186,A -130.6837,B 3.0793,C 0.277,E1 2.9789,E2 223.667} C_DIS
LIN {X -98.5163,Y -91.8973,Z 186,A -132.431,B 3.0795,C 0.2748,E1 2.9755,E2 225.4379} C_DIS
LIN {X -101.6028,Y -88.4728,Z 186,A -134.2377,B 3.0799,C 0.2701,E1 2.9722,E2 227.2246} C_DIS
LIN {X -103.9079,Y -85.754,Z 186,A -135.9482,B 3.0801,C 0.2679,E1 2.9691,E2 228.9595} C_DIS
LIN {X -106.7106,Y -82.2407,Z 186,A -137.9304,B 3.0804,C 0.2641,E1 2.9656,E2 230.9503} C_DIS
LIN {X -109.0019,Y -79.178,Z 186,A -139.6482,B 3.0807,C 0.2609,E1 2.9628,E2 232.6793} C_DIS
LIN {X -111.6967,Y -75.3289,Z 186,A -141.6349,B 3.0811,C 0.2564,E1 2.9596,E2 234.6639} C_DIS
LIN {X -113.9282,Y -71.909,Z 186,A -143.404,B 3.0814,C 0.2525,E1 2.9569,E2 236.4366} C_DIS
LIN {X -115.8989,Y -68.6885,Z 186,A -145.4316,B 3.0816,C 0.2504,E1 2.954,E2 238.517} C_DIS
LIN {X -117.6231,Y -65.6924,Z 186,A -146.6968,B 3.0819,C 0.2461,E1 2.9523,E2 239.7559} C_DIS
LIN {X -119.7961,Y -61.6379,Z 186,A -148.5495,B 3.0823,C 0.2409,E1 2.9499,E2 241.5947} C_DIS
LIN {X -120.9792,Y -59.2804,Z 186,A -149.8813,B 3.0825,C 0.2389,E1 2.9482,E2 242.9526} C_DIS
LIN {X -122.8795,Y -55.2332,Z 186,A -151.8288,B 3.0828,C 0.2343,E1 2.9459,E2 244.9051} C_DIS
LIN {X -124.2547,Y -52.0655,Z 186,A -153.3248,B 3.0831,C 0.2307,E1 2.9442,E2 246.4038} C_DIS
LIN {X -125.5085,Y -48.9659,Z 186,A -154.9708,B 3.0833,C 0.2279,E1 2.9425,E2 248.0774} C_DIS
LIN {X -126.8226,Y -45.4548,Z 186,A -156.4649,B 3.0836,C 0.2233,E1 2.9411,E2 249.5582} C_DIS
LIN {X -128.8587,Y -39.313,Z 186,A -159.3723,B 3.0841,C 0.2166,E1 2.9386,E2 252.4837} C_DIS
LIN {X -129.8133,Y -36.0364,Z 186,A -160.8753,B 3.0844,C 0.2129,E1 2.9374,E2 253.9925} C_DIS
LIN {X -130.65,Y -32.8744,Z 186,A -162.3515,B 3.0846,C 0.2094,E1 2.9364,E2 255.4786} C_DIS
LIN {X -131.5132,Y -29.2398,Z 186,A -164.1595,B 3.0849,C 0.2059,E1 2.9352,E2 257.3131} C_DIS
LIN {X -132.3067,Y -25.3974,Z 186,A -165.7585,B 3.0852,C 0.201,E1 2.9344,E2 258.9024} C_DIS
LIN {X -132.9394,Y -21.848,Z 186,A -167.481,B 3.0854,C 0.1975,E1 2.9335,E2 260.6477} C_DIS
LIN {X -133.5572,Y -17.6815,Z 186,A -169.2624,B 3.0857,C 0.1925,E1 2.9328,E2 262.4267} C_DIS
LIN {X -133.976,Y -14.1637,Z 186,A -170.8478,B 3.086,C 0.1885,E1 2.9323,E2 264.021} C_DIS
LIN {X -134.3475,Y -10.0473,Z 186,A -172.7104,B 3.0862,C 0.184,E1 2.9319,E2 265.8955} C_DIS
LIN {X -134.5593,Y -6.6317,Z 186,A -174.2078,B 3.0865,C 0.18,E1 2.9317,E2 267.3972} C_DIS
LIN {X -134.7,Y -2.4752,Z 186,A -176.116,B 3.0867,C 0.1755,E1 2.9315,E2 269.3214} C_DIS
LIN {X -134.7068,Y 2.0659,Z 186,A -178.1048,B 3.087,C 0.1703,E1 2.9315,E2 271.316} C_DIS
LIN {X -134.6027,Y 5.6976,Z 186,A -179.7763,B 3.0872,C 0.1664,E1 2.9317,E2 273.0021} C_DIS
LIN {X -134.3578,Y 9.906,Z 186,A 178.3745,B 3.0875,C 0.1615,E1 2.9321,E2 274.857} C_DIS
LIN {X -133.9845,Y 14.0855,Z 186,A 176.4958,B 3.0877,C 0.1569,E1 2.9326,E2 276.746} C_DIS
LIN {X -133.5635,Y 17.6332,Z 186,A 174.97,B 3.0879,C 0.1526,E1 2.9331,E2 278.2716} C_DIS
LIN {X -133.0193,Y 21.3668,Z 186,A 173.2487,B 3.0881,C 0.1486,E1 2.9338,E2 280.0061} C_DIS
LIN {X -132.3697,Y 25.0681,Z 186,A 170.6005,B 3.0881,C 0.1478,E1 2.9353,E2 282.78} C_DIS
LIN {X -130.9703,Y 31.5729,Z 186,A 168.4846,B 3.0887,C 0.1376,E1 2.9366,E2 284.8078} C_DIS
LIN {X -129.614,Y 36.7491,Z 186,A 166.2453,B 3.0889,C 0.1312,E1 2.9382,E2 287.0411} C_DIS
LIN {X -128.6964,Y 39.843,Z 186,A 164.6743,B 3.0891,C 0.1283,E1 2.9395,E2 288.6351} C_DIS
LIN {X -127.0443,Y 44.8363,Z 186,A 162.4939,B 3.0893,C 0.1221,E1 2.9414,E2 290.8071} C_DIS
LIN {X -126.052,Y 47.5504,Z 186,A 161.1301,B 3.0894,C 0.1194,E1 2.9428,E2 292.1862} C_DIS
LIN {X -124.7817,Y 50.7912,Z 186,A 159.5865,B 3.0895,C 0.1157,E1 2.9444,E2 293.7363} C_DIS
LIN {X -123.3268,Y 54.2326,Z 186,A 157.7194,B 3.0897,C 0.1127,E1 2.9465,E2 295.6358} C_DIS
LIN {X -121.1975,Y 58.8379,Z 186,A 155.7212,B 3.0899,C 0.1066,E1 2.9489,E2 297.6132} C_DIS
LIN {X -119.9582,Y 61.3196,Z 186,A 154.4862,B 3.0899,C 0.1039,E1 2.9504,E2 298.8538} C_DIS
LIN {X -118.3491,Y 64.3746,Z 186,A 152.8453,B 3.0901,C 0.1009,E1 2.9526,E2 300.5143} C_DIS
LIN {X -116.1871,Y 68.199,Z 186,A 150.9817,B 3.0902,C 0.0964,E1 2.9552,E2 302.3759} C_DIS
LIN {X -114.0539,Y 71.7099,Z 186,A 148.5545,B 3.0902,C 0.0948,E1 2.9589,E2 304.8827} C_DIS
LIN {X -111.3521,Y 75.8381,Z 186,A 147.0648,B 3.0905,C 0.0876,E1 2.9611,E2 306.2985} C_DIS
LIN {X -109.3665,Y 78.6744,Z 186,A 145.354,B 3.0905,C 0.0853,E1 2.9639,E2 308.0367} C_DIS
LIN {X -106.7254,Y 82.2216,Z 186,A 142.9922,B 3.0905,C 0.083,E1 2.968,E2 310.4541} C_DIS
LIN {X -103.9939,Y 85.6497,Z 186,A 141.6887,B 3.0908,C 0.0768,E1 2.9702,E2 311.6896} C_DIS
LIN {X -102.228,Y 87.7494,Z 186,A 139.8401,B 3.0908,C 0.0771,E1 2.9737,E2 313.6181} C_DIS
LIN {X -99.2616,Y 91.0917,Z 186,A 138.3085,B 3.0908,C 0.0717,E1 2.9765,E2 315.1047} C_DIS
LIN {X -94.7753,Y 95.751,Z 186,A 135.8034,B 3.091,C 0.0653,E1 2.9813,E2 317.5786} C_DIS
LIN {X -91.1409,Y 99.2163,Z 186,A 133.3031,B 3.091,C 0.0629,E1 2.9865,E2 320.1207} C_DIS
LIN {X -87.8146,Y 102.1722,Z 186,A 130.8812,B 3.091,C 0.0618,E1 2.9917,E2 322.6035} C_DIS
LIN {X -84.3952,Y 105.0145,Z 186,A 128.4547,B 3.0911,C 0.061,E1 2.9972,E2 325.091} C_DIS
LIN {X -78.9234,Y 109.1864,Z 186,A 126.4227,B 3.0913,C 0.0523,E1 3.0015,E2 327.0165} C_DIS
LIN {X -74.6474,Y 112.1533,Z 186,A 124.3142,B 3.0913,C 0.0484,E1 3.0063,E2 329.111} C_DIS
LIN {X -72.2623,Y 113.7053,Z 186,A 122.849,B 3.0913,C 0.0479,E1 3.0098,E2 330.6054} C_DIS
LIN {X -68.7957,Y 115.835,Z 186,A 121.1613,B 3.0913,C 0.0453,E1 3.0139,E2 332.2869} C_DIS
LIN {X -65.4521,Y 117.7566,Z 186,A 119.3988,B 3.0914,C 0.0438,E1 3.0182,E2 334.0626} C_DIS
LIN {X -60.6497,Y 120.2992,Z 186,A 117.1547,B 3.0914,C 0.0407,E1 3.0237,E2 336.2974} C_DIS
LIN {X -57.6532,Y 121.7635,Z 186,A 115.7175,B 3.0914,C 0.0392,E1 3.0273,E2 337.7359} C_DIS
LIN {X -54.3749,Y 123.2634,Z 186,A 113.6535,B 3.0914,C 0.0404,E1 3.0328,E2 339.8611} C_DIS
LIN {X -50.577,Y 124.8681,Z 186,A 111.4704,B 3.0914,C 0.0409,E1 3.0386,E2 342.0928} C_DIS
LIN {X -44.6491,Y 127.1094,Z 186,A 109.7417,B 3.0915,C 0.0335,E1 3.0428,E2 343.7073} C_DIS
LIN {X -39.2043,Y 128.8919,Z 186,A 107.2821,B 3.0915,C 0.0318,E1 3.0494,E2 346.1682} C_DIS
LIN {X -36.1381,Y 129.7849,Z 186,A 105.7818,B 3.0915,C 0.0316,E1 3.0534,E2 347.6844} C_DIS
LIN {X -32.8744,Y 130.65,Z 186,A 104.3395,B 3.0915,C 0.0308,E1 3.0573,E2 349.1266} C_DIS
LIN {X -29.8098,Y 131.383,Z 186,A 102.9854,B 3.0915,C 0.0302,E1 3.061,E2 350.4817} C_DIS
LIN {X -26.5836,Y 132.0738,Z 186,A 101.5565,B 3.0915,C 0.0297,E1 3.0649,E2 351.9128} C_DIS
LIN {X -23.4172,Y 132.6719,Z 186,A 100.2471,B 3.0915,C 0.0288,E1 3.0685,E2 353.2143} C_DIS
LIN {X -20.5437,Y 133.1468,Z 186,A 98.9393,B 3.0915,C 0.0288,E1 3.0722,E2 354.5296} C_DIS
LIN {X -16.7489,Y 133.6794,Z 186,A 96.8898,B 3.0915,C 0.031,E1 3.078,E2 356.6274} C_DIS
LIN {X -13.0304,Y 134.0909,Z 186,A 95.7675,B 3.0915,C 0.0279,E1 3.0809,E2 357.6941} C_DIS
LIN {X -9.6879,Y 134.3737,Z 186,A 94.3106,B 3.0915,C 0.0279,E1 3.085,E2 359.1539} C_DIS
LIN {X -6.1075,Y 134.5856,Z 186,A 92.6617,B 3.0915,C 0.0286,E1 3.0897,E2 360.8166} C_DIS
LIN {X -1.7457,Y 134.7122,Z 186,A 90.7995,B 3.0915,C 0.0288,E1 3.0949,E2 362.6788} C_DIS
LIN {X 1.3465,Y 134.7172,Z 186,A 89.4352,B 3.0915,C 0.0293,E1 3.0987,E2 364.0484} C_DIS
LIN {X 6.0502,Y 134.5883,Z 186,A 87.4505,B 3.0915,C 0.0296,E1 3.1042,E2 366.0303} C_DIS
LIN {X 10.294,Y 134.3295,Z 186,A 85.5575,B 3.0915,C 0.0308,E1 3.1095,E2 367.9325} C_DIS
LIN {X 14.9715,Y 133.8891,Z 186,A 83.6914,B 3.0915,C 0.0308,E1 3.1147,E2 369.7824} C_DIS
LIN {X 18.9591,Y 133.3817,Z 186,A 82.1179,B 3.0915,C 0.0306,E1 3.119,E2 371.3394} C_DIS
LIN {X 22.5738,Y 132.8183,Z 186,A 80.5784,B 3.0915,C 0.0314,E1 3.1232,E2 372.8765} C_DIS
LIN {X 26.5647,Y 132.0776,Z 186,A 78.8283,B 3.0915,C 0.0327,E1 3.128,E2 374.6289} C_DIS
LIN {X 30.1218,Y 131.3117,Z 186,A 77.2771,B 3.0915,C 0.0338,E1 3.1323,E2 376.1801} C_DIS
LIN {X 33.7432,Y 130.4295,Z 186,A 75.8092,B 3.0915,C 0.0342,E1 3.1362,E2 377.6338} C_DIS
LIN {X 37.0031,Y 129.543,Z 186,A 74.3753,B 3.0915,C 0.0355,E1 3.1401,E2 379.067} C_DIS
LIN {X 39.6525,Y 128.7547,Z 186,A 73.2268,B 3.0915,C 0.0363,E1 3.1431,E2 380.212} C_DIS
LIN {X 42.6846,Y 127.7814,Z 186,A 71.8566,B 3.0915,C 0.0378,E1 3.1468,E2 381.5838} C_DIS
LIN {X 45.8822,Y 126.6685,Z 186,A 70.4418,B 3.0915,C 0.0391,E1 3.1505,E2 382.9953} C_DIS
LIN {X 49.5954,Y 125.2638,Z 186,A 68.7998,B 3.0915,C 0.0407,E1 3.1548,E2 384.6317} C_DIS
LIN {X 52.153,Y 124.2182,Z 186,A 67.5977,B 3.0915,C 0.0422,E1 3.1579,E2 385.8367} C_DIS
LIN {X 55.5127,Y 122.7545,Z 186,A 66.1237,B 3.0915,C 0.0435,E1 3.1616,E2 387.3005} C_DIS
LIN {X 58.1327,Y 121.5343,Z 186,A 64.9217,B 3.0914,C 0.0449,E1 3.1647,E2 388.4991} C_DIS
LIN {X 61.0466,Y 120.0971,Z 186,A 63.5771,B 3.0914,C 0.0465,E1 3.168,E2 389.8392} C_DIS
LIN {X 66.1401,Y 117.3715,Z 186,A 61.2926,B 3.0914,C 0.0486,E1 3.1736,E2 392.1032} C_DIS
LIN {X 69.0371,Y 115.6911,Z 186,A 59.6796,B 3.0913,C 0.0523,E1 3.1775,E2 393.7385} C_DIS
LIN {X 72.6267,Y 113.4721,Z 186,A 57.9741,B 3.0913,C 0.0544,E1 3.1815,E2 395.4333} C_DIS
LIN {X 75.8279,Y 111.359,Z 186,A 56.3739,B 3.0912,C 0.0569,E1 3.1852,E2 397.0299} C_DIS
LIN {X 79.3708,Y 108.8622,Z 186,A 54.5213,B 3.0912,C 0.0601,E1 3.1894,E2 398.8836} C_DIS
LIN {X 82.9548,Y 106.1563,Z 186,A 52.6596,B 3.0911,C 0.0631,E1 3.1936,E2 400.7396} C_DIS
LIN {X 86.3954,Y 103.3753,Z 186,A 50.9075,B 3.0911,C 0.0655,E1 3.1973,E2 402.4765} C_DIS
LIN {X 89.5286,Y 100.6744,Z 186,A 48.9114,B 3.0909,C 0.0709,E1 3.2016,E2 404.501} C_DIS
LIN {X 92.1579,Y 98.2732,Z 186,A 47.6767,B 3.0909,C 0.0715,E1 3.204,E2 405.7025} C_DIS
LIN {X 95.346,Y 95.1829,Z 186,A 45.7579,B 3.0908,C 0.0756,E1 3.2078,E2 407.6252} C_DIS
LIN {X 98.2104,Y 92.2245,Z 186,A 44.207,B 3.0908,C 0.0775,E1 3.2108,E2 409.1524} C_DIS
LIN {X 101.167,Y 88.9714,Z 186,A 42.3734,B 3.0906,C 0.0812,E1 3.2142,E2 410.982} C_DIS
LIN {X 104.0189,Y 85.62,Z 186,A 40.5554,B 3.0906,C 0.0849,E1 3.2174,E2 412.794} C_DIS
LIN {X 106.7617,Y 82.1745,Z 186,A 38.7333,B 3.0904,C 0.0887,E1 3.2206,E2 414.6105} C_DIS
LIN {X 109.3615,Y 78.6814,Z 186,A 36.9319,B 3.0904,C 0.0925,E1 3.2235,E2 416.4062} C_DIS
LIN {X 111.8711,Y 75.07,Z 186,A 35.1899,B 3.0902,C 0.0957,E1 3.2262,E2 418.1333} C_DIS
LIN {X 114.0977,Y 71.6406,Z 186,A 33.5164,B 3.0902,C 0.0993,E1 3.2288,E2 419.7994} C_DIS
LIN {X 116.1886,Y 68.1966,Z 186,A 31.923,B 3.09,C 0.1024,E1 3.231,E2 421.3788} C_DIS
LIN {X 117.6039,Y 65.7266,Z 186,A 30.6787,B 3.09,C 0.1057,E1 3.2327,E2 422.6276} C_DIS
LIN {X 119.6923,Y 61.8418,Z 186,A 28.8481,B 3.0898,C 0.11,E1 3.2351,E2 424.4534} C_DIS
LIN {X 121.7247,Y 57.7344,Z 186,A 27.1256,B 3.0897,C 0.1128,E1 3.2372,E2 426.149} C_DIS
LIN {X 123.2214,Y 54.4688,Z 186,A 25.651,B 3.0895,C 0.1163,E1 3.2389,E2 427.6178} C_DIS
LIN {X 124.6596,Y 51.0942,Z 186,A 23.6879,B 3.0892,C 0.1242,E1 3.241,E2 429.6306} C_DIS
LIN {X 126.1536,Y 47.2789,Z 186,A 22.6922,B 3.0893,C 0.1217,E1 3.2419,E2 430.5359} C_DIS
LIN {X 126.9835,Y 45.0083,Z 186,A 21.4849,B 3.0891,C 0.1262,E1 3.2431,E2 431.7658} C_DIS
LIN {X 128.0579,Y 41.8541,Z 186,A 20.0363,B 3.089,C 0.1303,E1 3.2444,E2 433.2189} C_DIS
LIN {X 129.3021,Y 37.829,Z 186,A 18.4318,B 3.0888,C 0.1333,E1 3.2456,E2 434.8012} C_DIS
LIN {X 130.1881,Y 34.6572,Z 186,A 17.0785,B 3.0887,C 0.1367,E1 3.2466,E2 436.1494} C_DIS
LIN {X 130.9637,Y 31.6005,Z 186,A 15.8034,B 3.0886,C 0.1397,E1 3.2475,E2 437.4171} C_DIS
LIN {X 131.7188,Y 28.2888,Z 186,A 14.4066,B 3.0884,C 0.1432,E1 3.2483,E2 438.8088} C_DIS
LIN {X 132.4925,Y 24.4196,Z 186,A 12.6878,B 3.0882,C 0.1483,E1 3.2492,E2 440.5336} C_DIS
LIN {X 133.2109,Y 20.1294,Z 186,A 11.0859,B 3.088,C 0.151,E1 3.2499,E2 442.1058} C_DIS
LIN {X 133.6291,Y 17.1321,Z 186,A 9.7317,B 3.0878,C 0.1553,E1 3.2504,E2 443.4691} C_DIS
LIN {X 133.9771,Y 14.1536,Z 186,A 8.5412,B 3.0877,C 0.158,E1 3.2508,E2 444.6499} C_DIS
LIN {X 134.4078,Y 9.2206,Z 186,A 6.4906,B 3.0874,C 0.1634,E1 3.2512,E2 446.695} C_DIS
LIN {X 134.6173,Y 5.3239,Z 186,A 4.9684,B 3.0872,C 0.1667,E1 3.2514,E2 448.2011} C_DIS
LIN {X 134.7216,Y 0.7166,Z 186,A 3.0369,B 3.0869,C 0.172,E1 3.2515,E2 450.1303} C_DIS
LIN {X 134.6646,Y -3.9577,Z 186,A 1.2565,B 3.0867,C 0.1755,E1 3.2515,E2 451.8861} C_DIS
LIN {X 134.523,Y -7.3532,Z 186,A -0.3025,B 3.0864,C 0.1807,E1 3.2512,E2 453.4604} C_DIS
LIN {X 134.2286,Y -11.5267,Z 186,A -2.1109,B 3.0861,C 0.186,E1 3.2508,E2 455.2735} C_DIS
LIN {X 133.7234,Y -16.3813,Z 186,A -3.9405,B 3.0859,C 0.1894,E1 3.2502,E2 457.0738} C_DIS
LIN {X 133.1606,Y -20.4546,Z 186,A -5.5895,B 3.0857,C 0.1933,E1 3.2496,E2 458.7116} C_DIS
LIN {X 132.5087,Y -24.329,Z 186,A -7.2398,B 3.0854,C 0.1978,E1 3.2488,E2 460.3606} C_DIS
LIN {X 131.6854,Y -28.4435,Z 186,A -8.8263,B 3.0852,C 0.2008,E1 3.2479,E2 461.9234} C_DIS
LIN {X 130.8745,Y -31.9705,Z 186,A -10.3885,B 3.0849,C 0.2052,E1 3.2469,E2 463.4897} C_DIS
LIN {X 129.8354,Y -35.9574,Z 186,A -12.0695,B 3.0846,C 0.2093,E1 3.2457,E2 465.163} C_DIS
LIN {X 128.791,Y -39.5341,Z 186,A -13.4465,B 3.0845,C 0.2116,E1 3.2446,E2 466.515} C_DIS
LIN {X 125.8288,Y -48.1421,Z 186,A -17.6377,B 3.0835,C 0.2251,E1 3.2406,E2 470.7496} C_DIS
LIN {X 124.3422,Y -51.8561,Z 186,A -18.8179,B 3.0835,C 0.2245,E1 3.2395,E2 471.8653} C_DIS
LIN {X 122.8706,Y -55.2532,Z 186,A -20.3023,B 3.0833,C 0.2278,E1 3.2378,E2 473.3395} C_DIS
LIN {X 121.5307,Y -58.1405,Z 186,A -21.6927,B 3.083,C 0.2316,E1 3.2361,E2 474.7356} C_DIS
LIN {X 119.9872,Y -61.2626,Z 186,A -23.4639,B 3.0825,C 0.2382,E1 3.2338,E2 476.5448} C_DIS
LIN {X 118.0663,Y -64.8929,Z 186,A -24.8457,B 3.0825,C 0.2391,E1 3.2321,E2 477.8819} C_DIS
LIN {X 115.9402,Y -68.619,Z 186,A -26.6169,B 3.0821,C 0.2431,E1 3.2296,E2 479.6477} C_DIS
LIN {X 113.7895,Y -72.1288,Z 186,A -28.2318,B 3.0819,C 0.2461,E1 3.2272,E2 481.2467} C_DIS
LIN {X 111.646,Y -75.4038,Z 186,A -30.1789,B 3.0814,C 0.2528,E1 3.2241,E2 483.2311} C_DIS
LIN {X 109.3825,Y -78.652,Z 186,A -31.4951,B 3.0814,C 0.2533,E1 3.2221,E2 484.5019} C_DIS
LIN {X 106.7415,Y -82.2008,Z 186,A -33.3401,B 3.081,C 0.2573,E1 3.219,E2 486.3438} C_DIS
LIN {X 103.9677,Y -85.6817,Z 186,A -35.1312,B 3.0807,C 0.2606,E1 3.2158,E2 488.1233} C_DIS
LIN {X 101.1139,Y -89.0315,Z 186,A -37.0068,B 3.0804,C 0.2647,E1 3.2124,E2 490.001} C_DIS
LIN {X 97.7825,Y -92.6781,Z 186,A -39.087,B 3.08,C 0.269,E1 3.2084,E2 492.0803} C_DIS
LIN {X 95.2516,Y -95.2778,Z 186,A -40.4858,B 3.0798,C 0.2709,E1 3.2057,E2 493.4618} C_DIS
LIN {X 91.9648,Y -98.4534,Z 186,A -42.3733,B 3.0795,C 0.2744,E1 3.2019,E2 495.3437} C_DIS
LIN {X 89.4293,Y -100.7622,Z 186,A -43.7747,B 3.0793,C 0.2767,E1 3.199,E2 496.7388} C_DIS
LIN {X 85.6959,Y -103.956,Z 186,A -45.7419,B 3.0791,C 0.2796,E1 3.1948,E2 498.692} C_DIS
LIN {X 82.3257,Y -106.6448,Z 186,A -47.572,B 3.0787,C 0.283,E1 3.1908,E2 500.5231} C_DIS
LIN {X 78.6814,Y -109.3615,Z 186,A -49.2698,B 3.0787,C 0.2843,E1 3.187,E2 502.192} C_DIS
LIN {X 75.8519,Y -111.3427,Z 186,A -50.8655,B 3.0783,C 0.288,E1 3.1833,E2 503.8052} C_DIS
LIN {X 70.0555,Y -115.078,Z 186,A -54.3845,B 3.0774,C 0.2978,E1 3.1748,E2 507.4018} C_DIS
LIN {X 64.9969,Y -118.0087,Z 186,A -55.8825,B 3.0778,C 0.2931,E1 3.1715,E2 508.7743} C_DIS
LIN {X 60.8939,Y -120.1749,Z 186,A -57.9963,B 3.0774,C 0.2971,E1 3.1662,E2 510.9077} C_DIS
LIN {X 57.8454,Y -121.6716,Z 186,A -59.4372,B 3.0772,C 0.299,E1 3.1625,E2 512.3492} C_DIS
LIN {X 54.6532,Y -123.1389,Z 186,A -60.8049,B 3.0772,C 0.2999,E1 3.1591,E2 513.7015} C_DIS
LIN {X 51.618,Y -124.4416,Z 186,A -62.253,B 3.0769,C 0.302,E1 3.1553,E2 515.1563} C_DIS
LIN {X 48.5648,Y -125.6645,Z 186,A -63.5991,B 3.0769,C 0.3032,E1 3.1519,E2 516.4966} C_DIS
LIN {X 44.9836,Y -126.9924,Z 186,A -65.3551,B 3.0765,C 0.3061,E1 3.1472,E2 518.2707} C_DIS
LIN {X 41.2028,Y -128.267,Z 186,A -66.9024,B 3.0765,C 0.3066,E1 3.1431,E2 519.7997} C_DIS
LIN {X 37.8358,Y -129.3001,Z 186,A -68.3494,B 3.0764,C 0.3076,E1 3.1393,E2 521.241} C_DIS
LIN {X 34.5564,Y -130.215,Z 186,A -69.7365,B 3.0764,C 0.3085,E1 3.1356,E2 522.6212} C_DIS
LIN {X 31.067,Y -131.0923,Z 186,A -71.2601,B 3.0762,C 0.3097,E1 3.1314,E2 524.1449} C_DIS
LIN {X 28.1258,Y -131.754,Z 186,A -72.5085,B 3.0762,C 0.3104,E1 3.128,E2 525.3897} C_DIS
LIN {X 23.9947,Y -132.5686,Z 186,A -74.0948,B 3.0762,C 0.3101,E1 3.1237,E2 526.9505} C_DIS
LIN {X 21.0115,Y -133.0744,Z 186,A -75.6384,B 3.0759,C 0.3128,E1 3.1194,E2 528.5282} C_DIS
LIN {X 17.0371,Y -133.6416,Z 186,A -77.3385,B 3.0758,C 0.3137,E1 3.1147,E2 530.2283} C_DIS
LIN {X 12.4409,Y -134.1475,Z 186,A -79.5797,B 3.0755,C 0.3166,E1 3.1083,E2 532.5063} C_DIS
LIN {X 8.8446,Y -134.433,Z 186,A -80.6475,B 3.0758,C 0.3138,E1 3.1055,E2 533.5143} C_DIS
LIN {X 4.7479,Y -134.6398,Z 186,A -82.5516,B 3.0756,C 0.3154,E1 3.1001,E2 535.44} C_DIS
LIN {X 0.9798,Y -134.7172,Z 186,A -83.5203,B 3.076,C 0.3112,E1 3.0977,E2 536.3267} C_DIS
Enddeposition()
LIN {X 0.9798,Y -134.7172,Z 186,A -83.5203,B 3.076,C 0.3112,E1 3.0977,E2 536.3267} C_DIS
Startdeposition()
$VEL.CP = VEL_PRINT
LIN {X 1.6032,Y -135.6145,Z 186,A -83.0715,B 3.076,C 0.3115,E1 3.099,E2 535.8839} C_DIS
LIN {X 8.31,Y -135.3675,Z 186,A -80.2231,B 3.0761,C 0.3105,E1 3.1069,E2 533.0323} C_DIS
LIN {X 15.2055,Y -134.769,Z 186,A -77.377,B 3.0761,C 0.3098,E1 3.1148,E2 530.1952} C_DIS
LIN {X 18.973,Y -134.2887,Z 186,A -75.8486,B 3.0762,C 0.3096,E1 3.119,E2 528.6759} C_DIS
LIN {X 22.2716,Y -133.781,Z 186,A -74.1228,B 3.0766,C 0.3062,E1 3.1239,E2 526.9074} C_DIS
LIN {X 25.7292,Y -133.1595,Z 186,A -72.9285,B 3.0764,C 0.3075,E1 3.1271,E2 525.7506} C_DIS
LIN {X 29.8503,Y -132.2968,Z 186,A -71.1573,B 3.0766,C 0.3062,E1 3.1319,E2 523.9794} C_DIS
LIN {X 33.4455,Y -131.4334,Z 186,A -69.6729,B 3.0766,C 0.3055,E1 3.1359,E2 522.5043} C_DIS
LIN {X 37.3446,Y -130.3815,Z 186,A -67.8954,B 3.0768,C 0.3034,E1 3.1407,E2 520.7163} C_DIS
LIN {X 41.0628,Y -129.2564,Z 186,A -66.3678,B 3.0769,C 0.3027,E1 3.1448,E2 519.2026} C_DIS
LIN {X 46.1965,Y -127.5117,Z 186,A -64.105,B 3.0771,C 0.3005,E1 3.1507,E2 516.9421} C_DIS
LIN {X 50.1774,Y -125.9994,Z 186,A -62.2982,B 3.0773,C 0.2983,E1 3.1554,E2 515.1331} C_DIS
LIN {X 53.6675,Y -124.5516,Z 186,A -60.9505,B 3.0773,C 0.2984,E1 3.1588,E2 513.817} C_DIS
LIN {X 56.5938,Y -123.2499,Z 186,A -59.4113,B 3.0776,C 0.2951,E1 3.1628,E2 512.2523} C_DIS
LIN {X 59.5129,Y -121.8679,Z 186,A -57.9554,B 3.0779,C 0.2924,E1 3.1665,E2 510.7834} C_DIS
LIN {X 64.2352,Y -119.4473,Z 186,A -56.0727,B 3.0779,C 0.2924,E1 3.1711,E2 508.9465} C_DIS
LIN {X 67.1515,Y -117.8325,Z 186,A -54.1282,B 3.0785,C 0.2855,E1 3.176,E2 506.9301} C_DIS
LIN {X 70.7938,Y -115.681,Z 186,A -52.5228,B 3.0787,C 0.2843,E1 3.1797,E2 505.3474} C_DIS
LIN {X 73.7323,Y -113.8306,Z 186,A -51.3066,B 3.0787,C 0.2841,E1 3.1825,E2 504.1633} C_DIS
LIN {X 77.6682,Y -111.1825,Z 186,A -49.4787,B 3.0788,C 0.2822,E1 3.1867,E2 502.357} C_DIS
LIN {X 82.149,Y -107.9141,Z 186,A -47.0795,B 3.0793,C 0.2776,E1 3.1921,E2 499.9486} C_DIS
LIN {X 84.4773,Y -106.1009,Z 186,A -45.62,B 3.0797,C 0.2733,E1 3.1954,E2 498.4602} C_DIS
LIN {X 87.3421,Y -103.7556,Z 186,A -44.3705,B 3.0797,C 0.2733,E1 3.1979,E2 497.2509} C_DIS
LIN {X 90.435,Y -101.071,Z 186,A -42.3853,B 3.0802,C 0.2674,E1 3.2022,E2 495.2307} C_DIS
LIN {X 93.3477,Y -98.3879,Z 186,A -41.2011,B 3.0801,C 0.2686,E1 3.2044,E2 494.1096} C_DIS
LIN {X 97.6709,Y -94.0975,Z 186,A -38.576,B 3.0806,C 0.2628,E1 3.2096,E2 491.4756} C_DIS
LIN {X 100.2134,Y -91.3849,Z 186,A -36.8894,B 3.0809,C 0.2583,E1 3.2128,E2 489.7725} C_DIS
LIN {X 103.7317,Y -87.3706,Z 186,A -34.8761,B 3.0812,C 0.2556,E1 3.2164,E2 487.7892} C_DIS
LIN {X 106.7337,Y -83.6765,Z 186,A -32.9632,B 3.0815,C 0.252,E1 3.2198,E2 485.8875} C_DIS
LIN {X 109.4669,Y -80.068,Z 186,A -31.1862,B 3.0817,C 0.2488,E1 3.2227,E2 484.1266} C_DIS
LIN {X 114.2274,Y -73.1159,Z 186,A -27.6844,B 3.0824,C 0.2409,E1 3.2282,E2 480.6296} C_DIS
LIN {X 116.6414,Y -69.2003,Z 186,A -26.0731,B 3.0824,C 0.2393,E1 3.2304,E2 479.06} C_DIS
LIN {X 119.3644,Y -64.3897,Z 186,A -23.5061,B 3.0831,C 0.2312,E1 3.234,E2 476.4612} C_DIS
LIN {X 121.5183,Y -60.2216,Z 186,A -21.7381,B 3.0833,C 0.2283,E1 3.2362,E2 474.7193} C_DIS
LIN {X 122.983,Y -57.1712,Z 186,A -20.4429,B 3.0835,C 0.2259,E1 3.2377,E2 473.4404} C_DIS
LIN {X 124.3707,Y -54.086,Z 186,A -19.217,B 3.0836,C 0.2242,E1 3.2391,E2 472.2396} C_DIS
LIN {X 125.8183,Y -50.6266,Z 186,A -17.5309,B 3.084,C 0.219,E1 3.2409,E2 470.5391} C_DIS
LIN {X 127.236,Y -46.9546,Z 186,A -15.6027,B 3.0845,C 0.2119,E1 3.2428,E2 468.5754} C_DIS
LIN {X 128.3948,Y -43.6887,Z 186,A -14.2418,B 3.0847,C 0.209,E1 3.244,E2 467.2267} C_DIS
LIN {X 130.049,Y -38.4802,Z 186,A -12.265,B 3.0849,C 0.206,E1 3.2456,E2 465.291} C_DIS
LIN {X 131.0163,Y -35.0439,Z 186,A -10.8603,B 3.0851,C 0.2029,E1 3.2466,E2 463.8984} C_DIS
LIN {X 131.9083,Y -31.5219,Z 186,A -9.3621,B 3.0853,C 0.1991,E1 3.2476,E2 462.4038} C_DIS
LIN {X 132.835,Y -27.3557,Z 186,A -7.6537,B 3.0856,C 0.195,E1 3.2486,E2 460.7062} C_DIS
LIN {X 133.4705,Y -24.0631,Z 186,A -6.3533,B 3.0858,C 0.1923,E1 3.2493,E2 459.4196} C_DIS
LIN {X 133.9886,Y -20.988,Z 186,A -5.0759,B 3.086,C 0.189,E1 3.2499,E2 458.1464} C_DIS
LIN {X 134.4678,Y -17.6577,Z 186,A -3.8076,B 3.0861,C 0.1865,E1 3.2503,E2 456.8967} C_DIS
LIN {X 135.2092,Y -10.6033,Z 186,A -0.7227,B 3.0867,C 0.1773,E1 3.2512,E2 453.7986} C_DIS
LIN {X 135.4519,Y -6.7974,Z 186,A 0.7473,B 3.0868,C 0.1741,E1 3.2514,E2 452.3455} C_DIS
LIN {X 135.5878,Y -3.1297,Z 186,A 2.3431,B 3.0871,C 0.1693,E1 3.2515,E2 450.743} C_DIS
LIN {X 135.5497,Y 4.4997,Z 186,A 5.3963,B 3.0875,C 0.1619,E1 3.2515,E2 447.7094} C_DIS
LIN {X 135.0737,Y 12.2094,Z 186,A 8.4692,B 3.0879,C 0.1546,E1 3.2508,E2 444.6587} C_DIS
LIN {X 134.4391,Y 17.8766,Z 186,A 10.7779,B 3.0882,C 0.1489,E1 3.2501,E2 442.3613} C_DIS
LIN {X 133.8746,Y 21.7103,Z 186,A 12.3335,B 3.0883,C 0.1451,E1 3.2494,E2 440.815} C_DIS
LIN {X 133.2297,Y 25.3616,Z 186,A 13.821,B 3.0885,C 0.1415,E1 3.2486,E2 439.3366} C_DIS
LIN {X 132.3733,Y 29.5155,Z 186,A 15.5914,B 3.0887,C 0.1368,E1 3.2476,E2 437.5679} C_DIS
LIN {X 131.5399,Y 33.026,Z 186,A 16.9563,B 3.0888,C 0.1342,E1 3.2467,E2 436.2223} C_DIS
LIN {X 130.6713,Y 36.3098,Z 186,A 18.3087,B 3.089,C 0.1311,E1 3.2457,E2 434.8795} C_DIS
LIN {X 129.7157,Y 39.5876,Z 186,A 19.6786,B 3.089,C 0.1279,E1 3.2446,E2 433.5179} C_DIS
LIN {X 128.8389,Y 42.3571,Z 186,A 20.9219,B 3.0892,C 0.1244,E1 3.2436,E2 432.2721} C_DIS
LIN {X 127.6652,Y 45.7706,Z 186,A 22.1177,B 3.0892,C 0.1236,E1 3.2425,E2 431.1166} C_DIS
LIN {X 126.2495,Y 49.5434,Z 186,A 24.2336,B 3.0896,C 0.1151,E1 3.2403,E2 428.9484} C_DIS
LIN {X 124.3071,Y 54.2332,Z 186,A 26.122,B 3.0897,C 0.1119,E1 3.2383,E2 427.0911} C_DIS
LIN {X 122.1228,Y 58.9884,Z 186,A 28.206,B 3.0899,C 0.1075,E1 3.2358,E2 425.022} C_DIS
LIN {X 120.2582,Y 62.7009,Z 186,A 29.8398,B 3.0899,C 0.1042,E1 3.2338,E2 423.4026} C_DIS
LIN {X 118.0293,Y 66.8062,Z 186,A 32.0459,B 3.0902,C 0.0971,E1 3.2308,E2 421.167} C_DIS
LIN {X 116.2743,Y 69.8162,Z 186,A 33.2655,B 3.0902,C 0.0959,E1 3.229,E2 419.9783} C_DIS
LIN {X 114.1152,Y 73.2912,Z 186,A 34.8876,B 3.0904,C 0.0927,E1 3.2266,E2 418.3688} C_DIS
LIN {X 112.3698,Y 75.9398,Z 186,A 36.1906,B 3.0904,C 0.0898,E1 3.2246,E2 417.07} C_DIS
LIN {X 109.7115,Y 79.7323,Z 186,A 37.9956,B 3.0905,C 0.0867,E1 3.2217,E2 415.2831} C_DIS
LIN {X 107.3827,Y 82.8425,Z 186,A 39.6732,B 3.0906,C 0.0826,E1 3.2189,E2 413.6008} C_DIS
LIN {X 104.6245,Y 86.2995,Z 186,A 41.4774,B 3.0907,C 0.079,E1 3.2157,E2 411.804} C_DIS
LIN {X 101.6326,Y 89.8033,Z 186,A 43.3277,B 3.0908,C 0.0757,E1 3.2123,E2 409.9652} C_DIS
LIN {X 98.9332,Y 92.7696,Z 186,A 45.4405,B 3.091,C 0.0683,E1 3.2082,E2 407.8006} C_DIS
LIN {X 95.6094,Y 96.1908,Z 186,A 46.7107,B 3.091,C 0.0708,E1 3.2059,E2 406.6216} C_DIS
LIN {X 90.3368,Y 101.1589,Z 186,A 49.8962,B 3.091,C 0.0637,E1 3.1994,E2 403.4207} C_DIS
LIN {X 86.8473,Y 104.1708,Z 186,A 51.8073,B 3.0912,C 0.0603,E1 3.1953,E2 401.5139} C_DIS
LIN {X 83.3671,Y 106.9761,Z 186,A 53.6376,B 3.0912,C 0.0574,E1 3.1913,E2 399.6906} C_DIS
LIN {X 79.7039,Y 109.7321,Z 186,A 55.4806,B 3.0912,C 0.0548,E1 3.1872,E2 397.859} C_DIS
LIN {X 76.1394,Y 112.2348,Z 186,A 57.2839,B 3.0913,C 0.052,E1 3.183,E2 396.0601} C_DIS
LIN {X 72.2463,Y 114.7795,Z 186,A 59.1303,B 3.0913,C 0.0499,E1 3.1787,E2 394.2281} C_DIS
LIN {X 68.746,Y 116.9094,Z 186,A 60.8733,B 3.0913,C 0.0471,E1 3.1745,E2 392.4837} C_DIS
LIN {X 65.0315,Y 119.0157,Z 186,A 62.6388,B 3.0914,C 0.0448,E1 3.1702,E2 390.723} C_DIS
LIN {X 61.5699,Y 120.8405,Z 186,A 64.0597,B 3.0914,C 0.0444,E1 3.1668,E2 389.3303} C_DIS
LIN {X 58.754,Y 122.2348,Z 186,A 65.5197,B 3.0914,C 0.0415,E1 3.1631,E2 387.8544} C_DIS
LIN {X 55.7101,Y 123.652,Z 186,A 66.8189,B 3.0914,C 0.0407,E1 3.1598,E2 386.5699} C_DIS
LIN {X 52.6809,Y 124.9729,Z 186,A 68.2992,B 3.0915,C 0.0383,E1 3.156,E2 385.0796} C_DIS
LIN {X 49.3877,Y 126.31,Z 186,A 69.7095,B 3.0915,C 0.0373,E1 3.1523,E2 383.6805} C_DIS
LIN {X 46.3868,Y 127.4431,Z 186,A 70.9712,B 3.0915,C 0.0366,E1 3.1491,E2 382.4304} C_DIS
LIN {X 43.0943,Y 128.5934,Z 186,A 72.4144,B 3.0915,C 0.0353,E1 3.1453,E2 380.991} C_DIS
LIN {X 39.8193,Y 129.6448,Z 186,A 73.9127,B 3.0915,C 0.0336,E1 3.1412,E2 379.4876} C_DIS
LIN {X 36.7382,Y 130.5514,Z 186,A 75.2935,B 3.0915,C 0.0322,E1 3.1375,E2 378.1042} C_DIS
LIN {X 32.7063,Y 131.621,Z 186,A 77.0989,B 3.0915,C 0.0305,E1 3.1326,E2 376.2942} C_DIS
LIN {X 28.7121,Y 132.548,Z 186,A 78.7019,B 3.0915,C 0.0301,E1 3.1283,E2 374.7071} C_DIS
LIN {X 24.941,Y 133.3101,Z 186,A 80.3999,B 3.0916,C 0.0285,E1 3.1236,E2 373.001} C_DIS
LIN {X 20.7899,Y 134.0193,Z 186,A 82.0161,B 3.0916,C 0.0287,E1 3.1192,E2 371.4048} C_DIS
LIN {X 17.4646,Y 134.4931,Z 186,A 83.5104,B 3.0916,C 0.0274,E1 3.115,E2 369.902} C_DIS
LIN {X 9.8677,Y 135.2629,Z 186,A 86.7106,B 3.0916,C 0.0264,E1 3.1062,E2 366.7062} C_DIS
LIN {X 5.6981,Y 135.5033,Z 186,A 88.4966,B 3.0916,C 0.0258,E1 3.1012,E2 364.9183} C_DIS
LIN {X 2.8056,Y 135.5945,Z 186,A 89.9125,B 3.0916,C 0.0243,E1 3.0971,E2 363.4797} C_DIS
LIN {X -4.3208,Y 135.5547,Z 186,A 92.757,B 3.0916,C 0.0251,E1 3.0892,E2 360.6565} C_DIS
LIN {X -8.4406,Y 135.3595,Z 186,A 94.3769,B 3.0916,C 0.026,E1 3.0848,E2 359.0521} C_DIS
LIN {X -12.3808,Y 135.0572,Z 186,A 96.5145,B 3.0916,C 0.0232,E1 3.0787,E2 356.8591} C_DIS
LIN {X -16.2889,Y 134.6407,Z 186,A 97.8343,B 3.0916,C 0.0257,E1 3.0751,E2 355.581} C_DIS
LIN {X -20.5374,Y 134.0583,Z 186,A 99.5498,B 3.0916,C 0.0268,E1 3.0704,E2 353.878} C_DIS
LIN {X -23.5297,Y 133.5659,Z 186,A 100.934,B 3.0916,C 0.0266,E1 3.0665,E2 352.4821} C_DIS
LIN {X -26.9639,Y 132.9147,Z 186,A 102.3205,B 3.0916,C 0.0278,E1 3.0628,E2 351.1072} C_DIS
LIN {X -30.4144,Y 132.1679,Z 186,A 103.8786,B 3.0916,C 0.0282,E1 3.0585,E2 349.5419} C_DIS
LIN {X -34.5071,Y 131.1595,Z 186,A 105.6869,B 3.0916,C 0.029,E1 3.0536,E2 347.7313} C_DIS
LIN {X -38.5071,Y 130.0412,Z 186,A 107.4036,B 3.0916,C 0.0304,E1 3.049,E2 346.0203} C_DIS
LIN {X -42.4842,Y 128.7965,Z 186,A 109.2258,B 3.0916,C 0.0314,E1 3.0441,E2 344.1917} C_DIS
LIN {X -45.9869,Y 127.5873,Z 186,A 111.4482,B 3.0916,C 0.029,E1 3.0381,E2 341.8909} C_DIS
LIN {X -50.8012,Y 125.7479,Z 186,A 113.0389,B 3.0916,C 0.0343,E1 3.0341,E2 340.3725} C_DIS
LIN {X -54.6887,Y 124.1088,Z 186,A 114.9347,B 3.0916,C 0.0355,E1 3.0292,E2 338.4643} C_DIS
LIN {X -58.2198,Y 122.49,Z 186,A 116.4394,B 3.0916,C 0.038,E1 3.0255,E2 336.977} C_DIS
LIN {X -60.4969,Y 121.3825,Z 186,A 118.2537,B 3.0916,C 0.0354,E1 3.0207,E2 335.0735} C_DIS
LIN {X -65.1917,Y 118.9284,Z 186,A 119.9722,B 3.0915,C 0.0409,E1 3.0166,E2 333.4195} C_DIS
LIN {X -69.129,Y 116.6839,Z 186,A 121.9362,B 3.0915,C 0.0431,E1 3.0119,E2 331.4509} C_DIS
LIN {X -72.8979,Y 114.3669,Z 186,A 124.139,B 3.0915,C 0.0441,E1 3.0066,E2 329.209} C_DIS
LIN {X -76.0755,Y 112.278,Z 186,A 125.467,B 3.0914,C 0.0479,E1 3.0036,E2 327.9159} C_DIS
LIN {X -80.063,Y 109.4707,Z 186,A 128.304,B 3.0914,C 0.0474,E1 2.997,E2 324.9859} C_DIS
LIN {X -84.7274,Y 105.9013,Z 186,A 130.0323,B 3.0913,C 0.0551,E1 2.9934,E2 323.3511} C_DIS
LIN {X -87.8275,Y 103.3448,Z 186,A 131.8885,B 3.0913,C 0.0573,E1 2.9894,E2 321.477} C_DIS
LIN {X -91.335,Y 100.2587,Z 186,A 133.9099,B 3.0911,C 0.0607,E1 2.9851,E2 319.4513} C_DIS
LIN {X -94.4848,Y 97.2958,Z 186,A 135.5898,B 3.0911,C 0.0648,E1 2.9818,E2 317.7905} C_DIS
LIN {X -96.2597,Y 95.5398,Z 186,A 137.0299,B 3.0911,C 0.0651,E1 2.9789,E2 316.3044} C_DIS
LIN {X -99.8049,Y 91.8303,Z 186,A 138.9795,B 3.0909,C 0.0704,E1 2.9752,E2 314.383} C_DIS
LIN {X -103.9399,Y 87.1225,Z 186,A 142.3294,B 3.0909,C 0.073,E1 2.9689,E2 310.9495} C_DIS
LIN {X -106.7635,Y 83.6385,Z 186,A 143.9249,B 3.0908,C 0.0783,E1 2.9662,E2 309.392} C_DIS
LIN {X -109.5598,Y 79.9416,Z 186,A 146.1383,B 3.0907,C 0.0816,E1 2.9625,E2 307.149} C_DIS
LIN {X -111.5885,Y 77.0844,Z 186,A 147.6629,B 3.0906,C 0.0848,E1 2.9601,E2 305.6201} C_DIS
LIN {X -113.5048,Y 74.2338,Z 186,A 149.0027,B 3.0905,C 0.0887,E1 2.9581,E2 304.295} C_DIS
LIN {X -116.0549,Y 70.1789,Z 186,A 151.0079,B 3.0903,C 0.0935,E1 2.9551,E2 302.2936} C_DIS
LIN {X -118.1287,Y 66.6294,Z 186,A 152.8083,B 3.0903,C 0.0975,E1 2.9526,E2 300.4868} C_DIS
LIN {X -119.9337,Y 63.3189,Z 186,A 154.3695,B 3.0901,C 0.1015,E1 2.9505,E2 298.9306} C_DIS
LIN {X -121.4912,Y 60.2765,Z 186,A 155.9641,B 3.09,C 0.1046,E1 2.9485,E2 297.3186} C_DIS
LIN {X -122.9417,Y 57.2604,Z 186,A 157.9688,B 3.09,C 0.1059,E1 2.9461,E2 295.2421} C_DIS
LIN {X -124.8621,Y 52.946,Z 186,A 159.5358,B 3.0897,C 0.1127,E1 2.9444,E2 293.7296} C_DIS
LIN {X -126.254,Y 49.5319,Z 186,A 161.1394,B 3.0895,C 0.1165,E1 2.9427,E2 292.1216} C_DIS
LIN {X -127.7441,Y 45.5519,Z 186,A 163.5018,B 3.0895,C 0.1192,E1 2.9404,E2 289.6902} C_DIS
LIN {X -129.1249,Y 41.4744,Z 186,A 164.6316,B 3.0892,C 0.1266,E1 2.9395,E2 288.6472} C_DIS
LIN {X -130.6503,Y 36.3846,Z 186,A 167.2755,B 3.089,C 0.1312,E1 2.9374,E2 285.9557} C_DIS
LIN {X -131.7545,Y 32.1598,Z 186,A 169.6565,B 3.0888,C 0.1342,E1 2.9358,E2 283.5092} C_DIS
LIN {X -132.6957,Y 28.028,Z 186,A 171.2137,B 3.0886,C 0.14,E1 2.9349,E2 281.9825} C_DIS
LIN {X -133.5016,Y 23.8891,Z 186,A 172.9117,B 3.0883,C 0.1453,E1 2.934,E2 280.2962} C_DIS
LIN {X -134.0535,Y 20.5688,Z 186,A 174.4407,B 3.0882,C 0.1488,E1 2.9333,E2 278.7548} C_DIS
LIN {X -134.6156,Y 16.4989,Z 186,A 176.2795,B 3.0879,C 0.1533,E1 2.9327,E2 276.9044} C_DIS
LIN {X -135.0126,Y 12.8463,Z 186,A 177.8573,B 3.0877,C 0.1576,E1 2.9322,E2 275.3244} C_DIS
LIN {X -135.3408,Y 8.7443,Z 186,A 179.7226,B 3.0875,C 0.162,E1 2.9318,E2 273.4444} C_DIS
LIN {X -135.5274,Y 5.0779,Z 186,A -178.6699,B 3.0873,C 0.1662,E1 2.9316,E2 271.8309} C_DIS
LIN {X -135.6219,Y 0.6639,Z 186,A -176.7393,B 3.087,C 0.1712,E1 2.9316,E2 269.8933} C_DIS
LIN {X -135.5837,Y -3.2759,Z 186,A -174.9241,B 3.0868,C 0.1753,E1 2.9316,E2 268.0603} C_DIS
LIN {X -135.4375,Y -7.0843,Z 186,A -173.3046,B 3.0865,C 0.1798,E1 2.9318,E2 266.4405} C_DIS
LIN {X -135.1651,Y -11.1306,Z 186,A -171.4817,B 3.0863,C 0.1842,E1 2.9322,E2 264.6049} C_DIS
LIN {X -134.8176,Y -14.7533,Z 186,A -169.8308,B 3.086,C 0.1881,E1 2.9327,E2 262.9406} C_DIS
LIN {X -134.3029,Y -18.8739,Z 186,A -168.0216,B 3.0857,C 0.1928,E1 2.9334,E2 261.1255} C_DIS
LIN {X -133.8056,Y -22.1241,Z 186,A -166.6903,B 3.0855,C 0.1969,E1 2.934,E2 259.8023} C_DIS
LIN {X -133.2207,Y -25.4089,Z 186,A -165.1303,B 3.0853,C 0.2002,E1 2.9348,E2 258.224} C_DIS
LIN {X -132.4216,Y -29.2979,Z 186,A -163.2444,B 3.085,C 0.204,E1 2.9359,E2 256.3126} C_DIS
LIN {X -131.5978,Y -32.7978,Z 186,A -161.725,B 3.0847,C 0.2081,E1 2.9369,E2 254.7939} C_DIS
LIN {X -130.6986,Y -36.2122,Z 186,A -160.1866,B 3.0845,C 0.212,E1 2.938,E2 253.2503} C_DIS
LIN {X -128.9706,Y -41.9555,Z 186,A -157.2528,B 3.0841,C 0.2172,E1 2.9405,E2 250.2665} C_DIS
LIN {X -127.8907,Y -45.1425,Z 186,A -156.0961,B 3.0838,C 0.222,E1 2.9415,E2 249.1445} C_DIS
LIN {X -126.5189,Y -48.8504,Z 186,A -154.4502,B 3.0834,C 0.2264,E1 2.9431,E2 247.5025} C_DIS
LIN {X -125.2483,Y -52.0213,Z 186,A -152.8053,B 3.0832,C 0.2293,E1 2.9449,E2 245.8323} C_DIS
LIN {X -123.8209,Y -55.3324,Z 186,A -151.3701,B 3.0829,C 0.2336,E1 2.9465,E2 244.4091} C_DIS
LIN {X -122.523,Y -58.1507,Z 186,A -149.8366,B 3.0827,C 0.2359,E1 2.9483,E2 242.8476} C_DIS
LIN {X -120.5648,Y -62.1113,Z 186,A -147.9069,B 3.0824,C 0.2403,E1 2.9508,E2 240.9105} C_DIS
LIN {X -119.0582,Y -64.9536,Z 186,A -146.5682,B 3.0821,C 0.2437,E1 2.9525,E2 239.575} C_DIS
LIN {X -116.7145,Y -69.0778,Z 186,A -144.2986,B 3.0818,C 0.2474,E1 2.9558,E2 237.2718} C_DIS
LIN {X -114.316,Y -72.9774,Z 186,A -142.3629,B 3.0815,C 0.2518,E1 2.9586,E2 235.3365} C_DIS
LIN {X -112.0307,Y -76.4401,Z 186,A -140.463,B 3.0812,C 0.2552,E1 2.9616,E2 233.4181} C_DIS
LIN {X -109.457,Y -80.0816,Z 186,A -138.5113,B 3.0809,C 0.2591,E1 2.9648,E2 231.458} C_DIS
LIN {X -106.6544,Y -83.7775,Z 186,A -136.5162,B 3.0805,C 0.2631,E1 2.9682,E2 229.4588} C_DIS
LIN {X -103.8592,Y -87.2186,Z 186,A -134.6139,B 3.0802,C 0.2669,E1 2.9716,E2 227.553} C_DIS
LIN {X -101.1223,Y -90.3776,Z 186,A -132.393,B 3.0801,C 0.2683,E1 2.9758,E2 225.2731} C_DIS
LIN {X -98.423,Y -93.3105,Z 186,A -130.9949,B 3.0797,C 0.273,E1 2.9784,E2 223.9127} C_DIS
LIN {X -95.4344,Y -96.3646,Z 186,A -129.0716,B 3.0794,C 0.2759,E1 2.9823,E2 221.9742} C_DIS
LIN {X -92.063,Y -99.591,Z 186,A -127.0582,B 3.0791,C 0.2793,E1 2.9864,E2 219.9556} C_DIS
LIN {X -88.6677,Y -102.6251,Z 186,A -125.0949,B 3.0788,C 0.2824,E1 2.9905,E2 217.9872} C_DIS
LIN {X -85.1352,Y -105.5738,Z 186,A -123.1252,B 3.0785,C 0.2855,E1 2.9948,E2 216.0143} C_DIS
LIN {X -81.5544,Y -108.3639,Z 186,A -121.1552,B 3.0783,C 0.2883,E1 2.9992,E2 214.0375} C_DIS
LIN {X -77.8555,Y -111.0518,Z 186,A -119.1547,B 3.078,C 0.2909,E1 3.0037,E2 212.0281} C_DIS
LIN {X -74.2137,Y -113.518,Z 186,A -117.2585,B 3.0778,C 0.2934,E1 3.0082,E2 210.1267} C_DIS
LIN {X -70.4573,Y -115.8866,Z 186,A -115.5773,B 3.0775,C 0.297,E1 3.0121,E2 208.471} C_DIS
LIN {X -68.2763,Y -117.1847,Z 186,A -114.2101,B 3.0775,C 0.2967,E1 3.0155,E2 207.065} C_DIS
LIN {X -64.1858,Y -119.4739,Z 186,A -112.1891,B 3.0773,C 0.2989,E1 3.0204,E2 205.0385} C_DIS
LIN {X -60.2501,Y -121.5042,Z 186,A -110.4111,B 3.077,C 0.3015,E1 3.0249,E2 203.2724} C_DIS
LIN {X -57.1275,Y -123.0032,Z 186,A -108.9589,B 3.0769,C 0.3031,E1 3.0285,E2 201.8215} C_DIS
LIN {X -54.0689,Y -124.3781,Z 186,A -107.5538,B 3.0767,C 0.3046,E1 3.0321,E2 200.4177} C_DIS
LIN {X -50.9906,Y -125.6716,Z 186,A -106.0864,B 3.0767,C 0.3056,E1 3.0359,E2 198.9426} C_DIS
LIN {X -48.1148,Y -126.8014,Z 186,A -104.6801,B 3.0766,C 0.3061,E1 3.0396,E2 197.5228} C_DIS
LIN {X -44.971,Y -127.9502,Z 186,A -103.2176,B 3.0765,C 0.3069,E1 3.0435,E2 196.0535} C_DIS
LIN {X -41.453,Y -129.1317,Z 186,A -101.7135,B 3.0763,C 0.3084,E1 3.0475,E2 194.5574} C_DIS
LIN {X -38.1996,Y -130.1312,Z 186,A -100.2726,B 3.0763,C 0.3094,E1 3.0513,E2 193.1157} C_DIS
LIN {X -34.9621,Y -131.0381,Z 186,A -98.832,B 3.0762,C 0.31,E1 3.0552,E2 191.6721} C_DIS
LIN {X -31.8225,Y -131.8358,Z 186,A -97.4046,B 3.0762,C 0.3104,E1 3.0591,E2 190.2365} C_DIS
LIN {X -27.804,Y -132.7437,Z 186,A -95.5697,B 3.0762,C 0.3105,E1 3.0642,E2 188.3886} C_DIS
LIN {X -24.1428,Y -133.4562,Z 186,A -94.0942,B 3.076,C 0.3117,E1 3.0682,E2 186.9257} C_DIS
LIN {X -20.8905,Y -134.0037,Z 186,A -92.7078,B 3.076,C 0.3122,E1 3.072,E2 185.5398} C_DIS
LIN {X -12.7786,Y -135.0191,Z 186,A -89.2139,B 3.076,C 0.3125,E1 3.0817,E2 182.0393} C_DIS
LIN {X -8.7389,Y -135.3411,Z 186,A -87.2512,B 3.0761,C 0.3107,E1 3.0873,E2 180.0427} C_DIS
LIN {X -3.9772,Y -135.5642,Z 186,A -84.8062,B 3.0764,C 0.3075,E1 3.0943,E2 177.5393} C_DIS
LIN {X 0.9717,Y -135.6088,Z 186,A -84.5624,B 3.0751,C 0.3205,E1 3.0944,E2 177.5382} C_DIS
Enddeposition()
LIN {X 0.9717,Y -135.6088,Z 186,A -84.5628,B 3.0751,C 0.3205,E1 3.0944,E2 177.5388} C_DIS
Startdeposition()
$VEL.CP = VEL_PRINT
LIN {X -0.3966,Y -136.5222,Z 186,A -85.0346,B 2.9885,C 0.3183,E1 3.0064,E2 178.0539} C_DIS
LIN {X -4.9292,Y -136.4338,Z 186,A -86.2544,B 2.9889,C 0.3137,E1 3.0032,E2 179.1845} C_DIS
Enddeposition()
END
